REGION Network 5: Special Function Buttons Operator Control Allowed
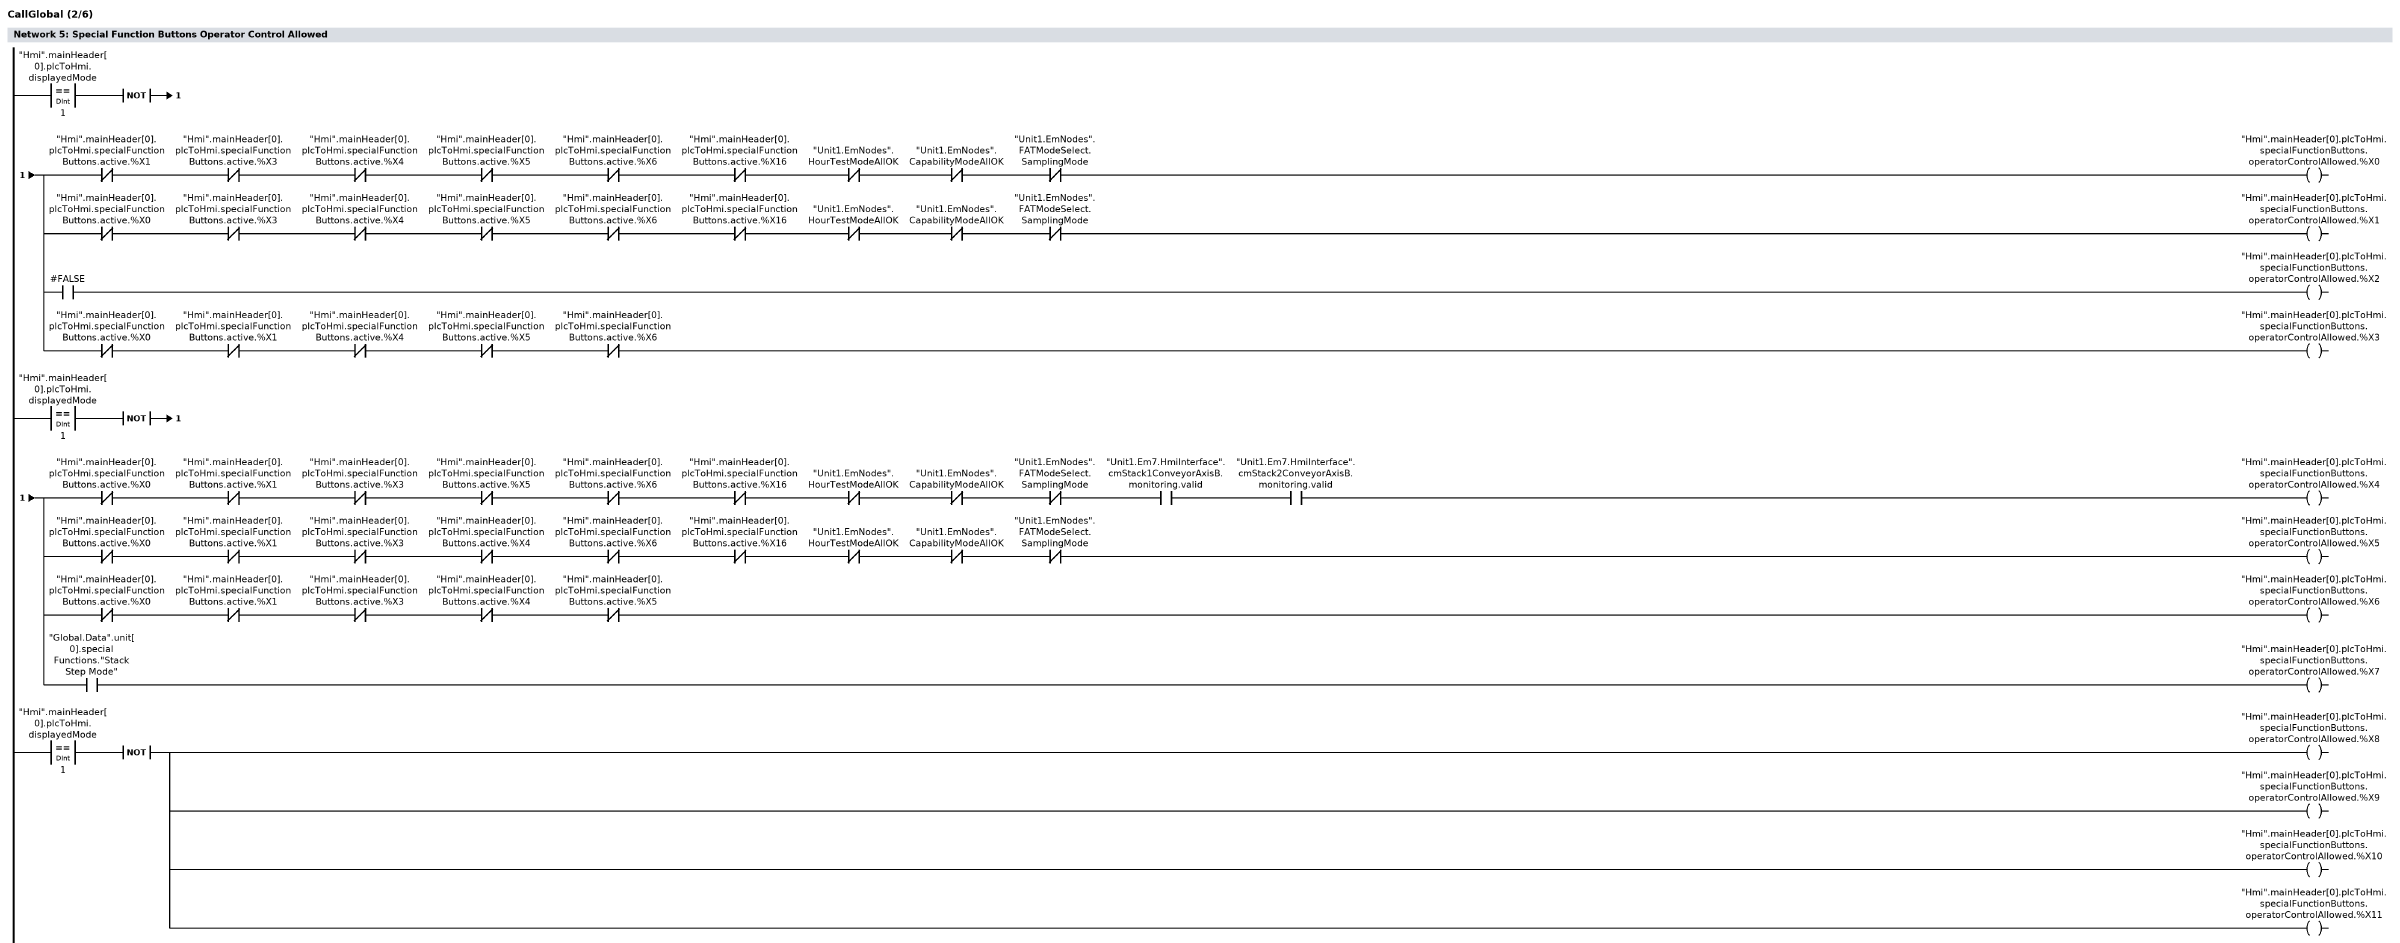
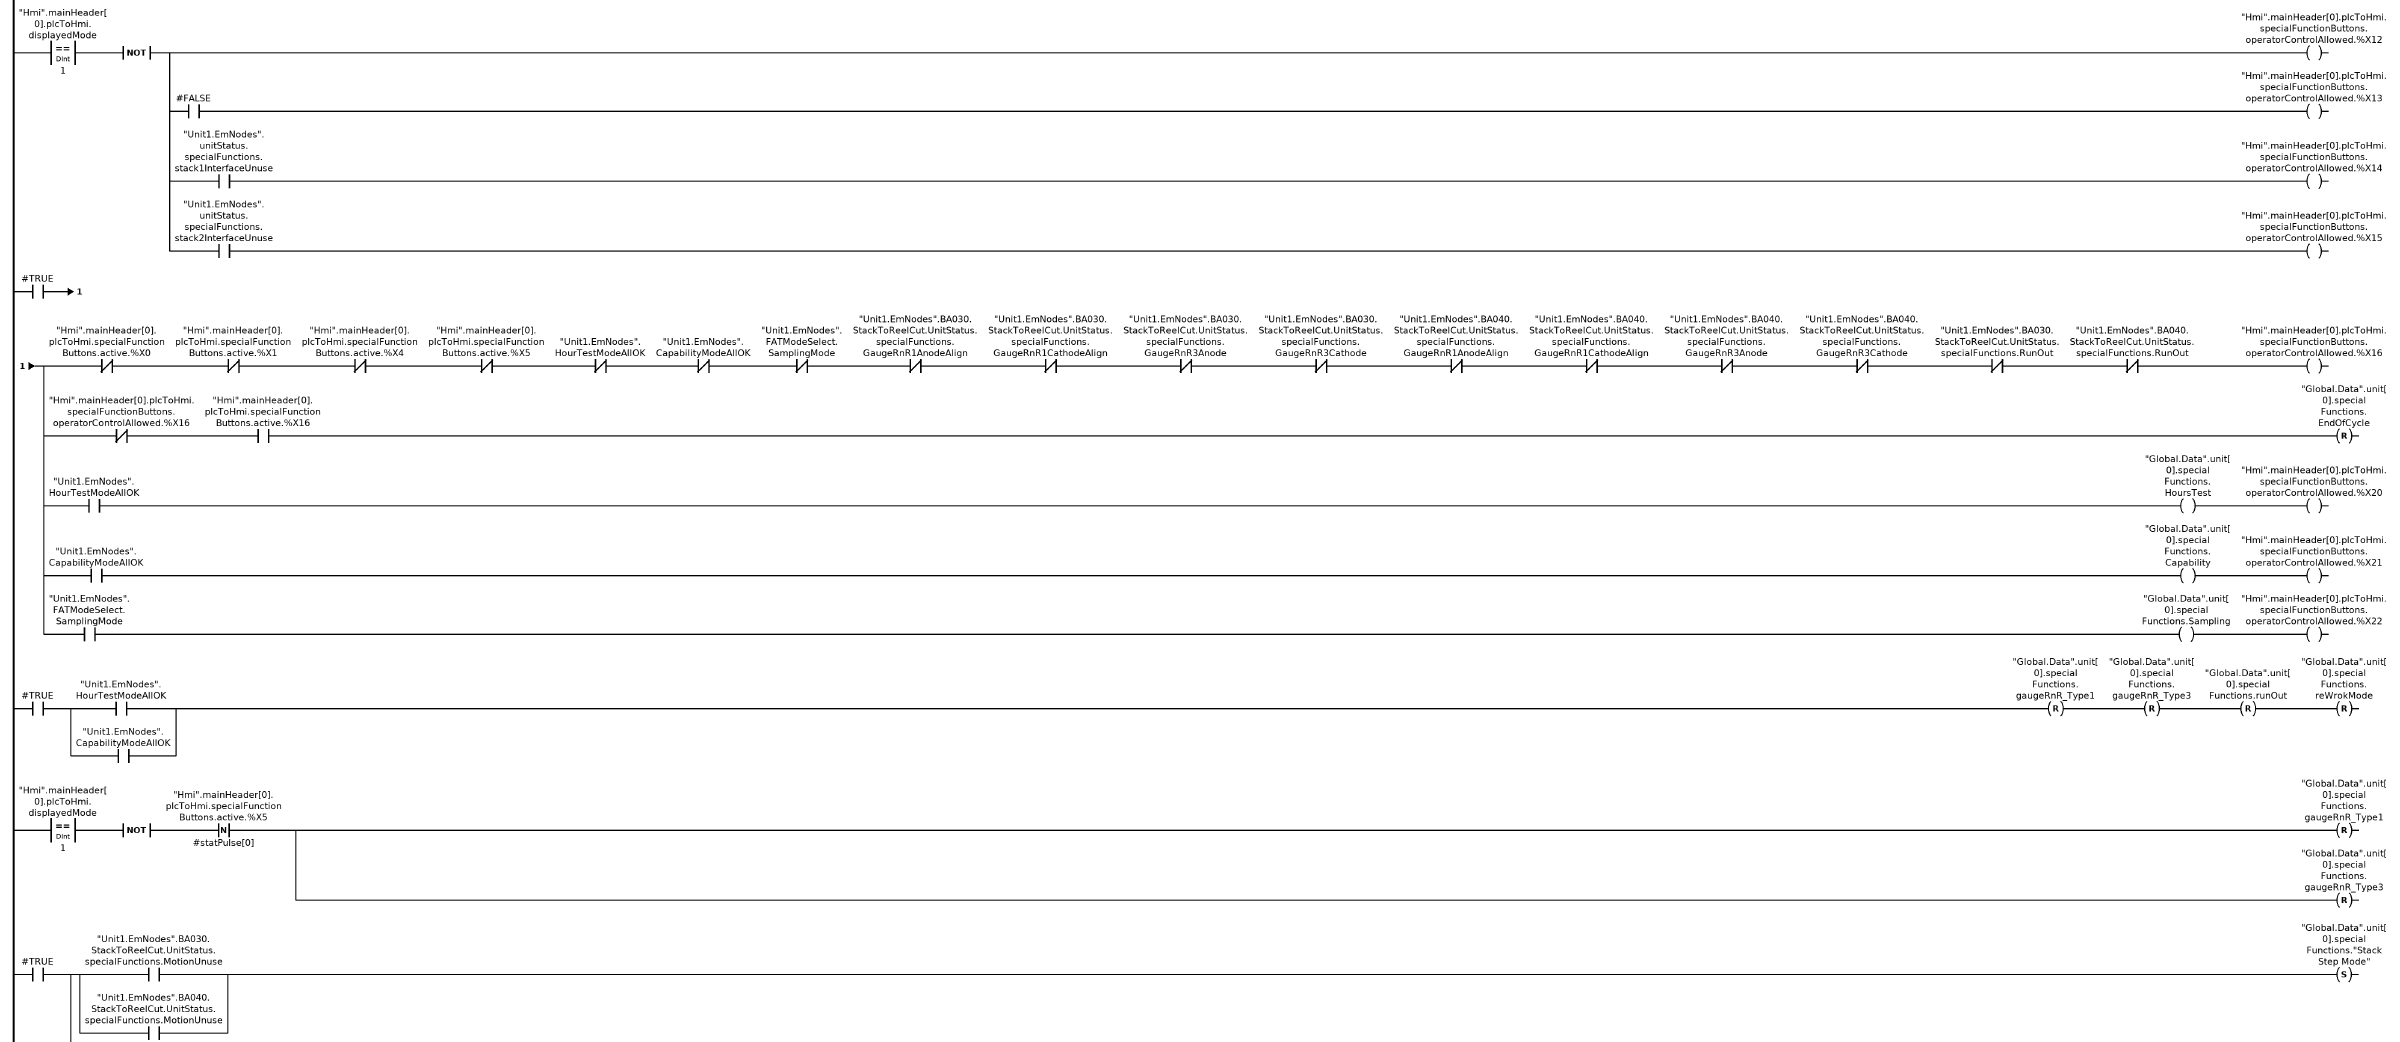
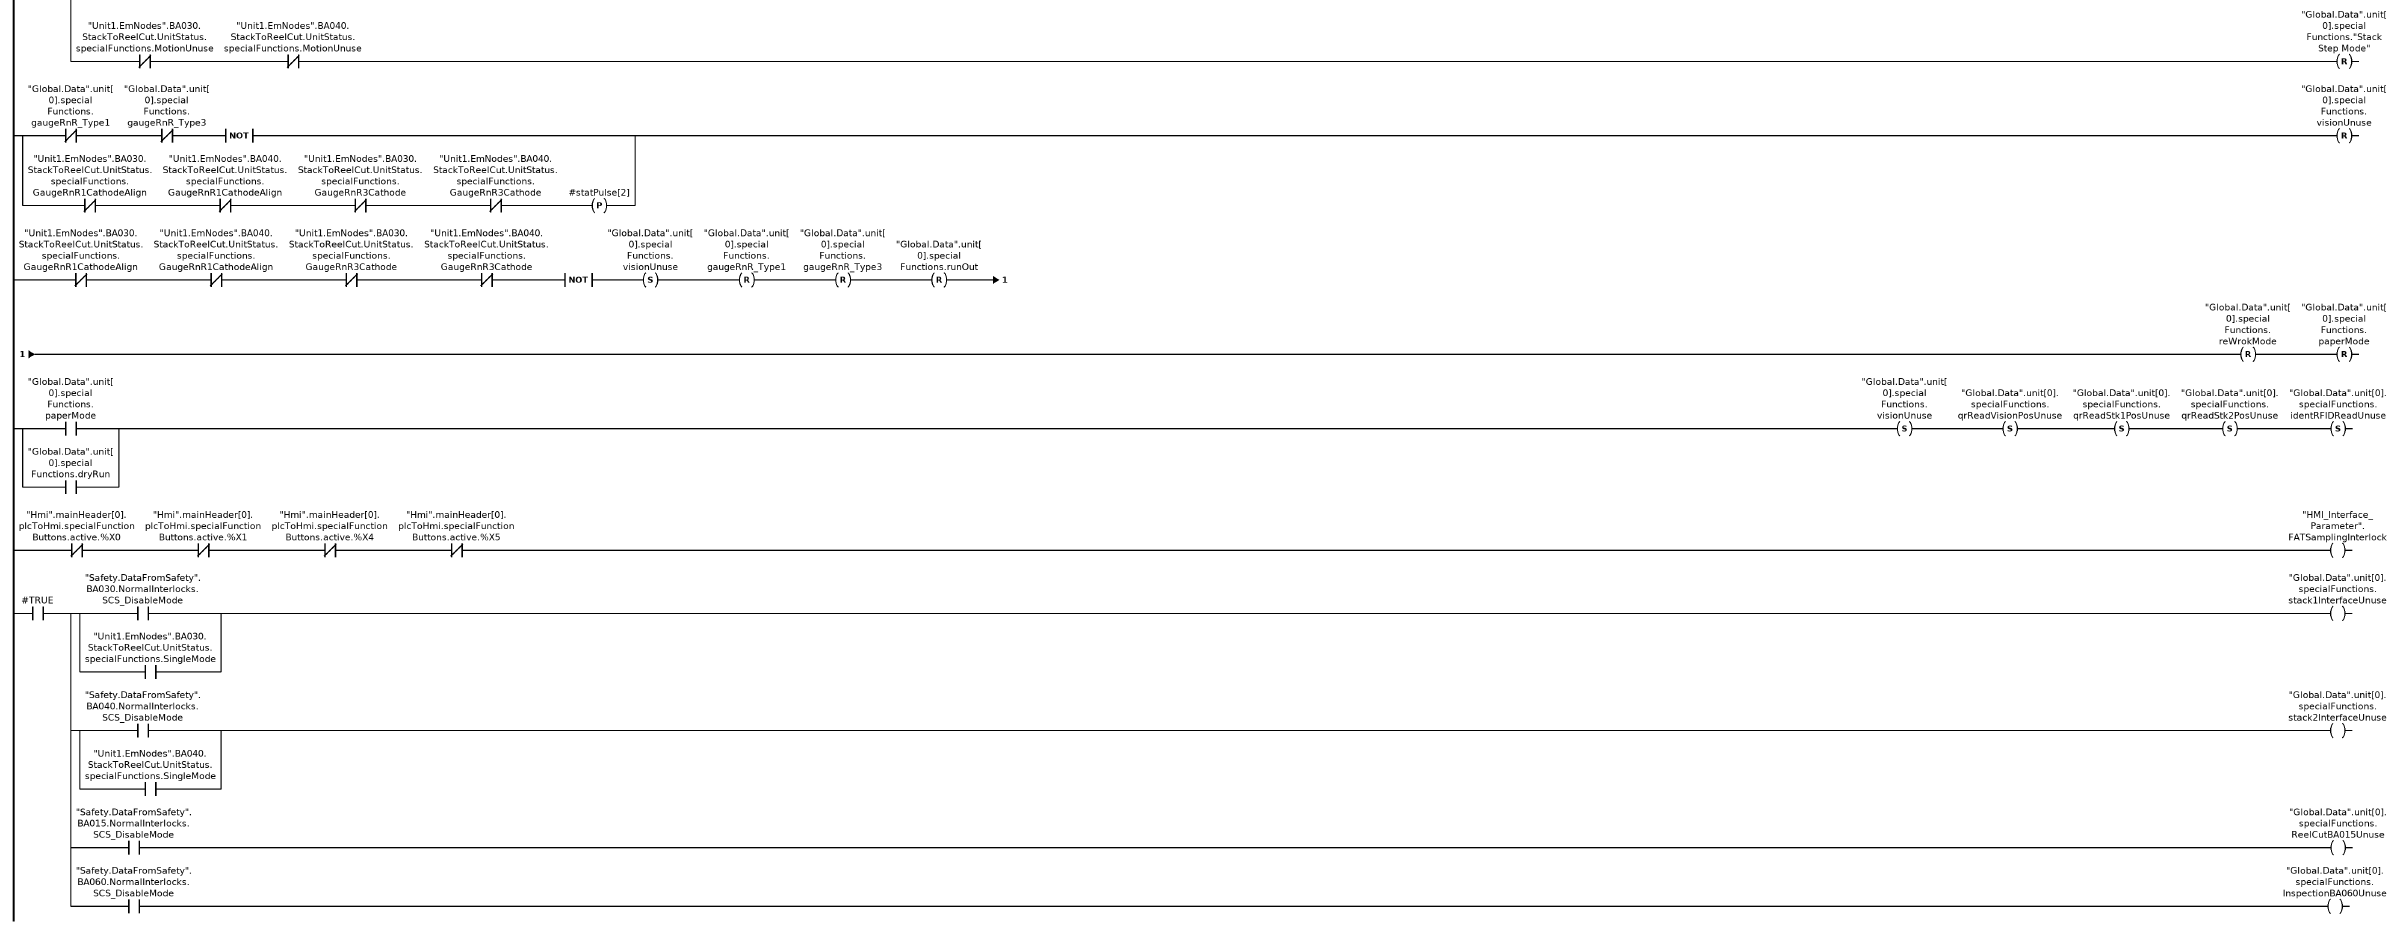
   RUNG wire#powerrail
      { S7_Templates := "SrcType := DInt" } EQ_Contact(in1 := "Hmi".mainHeader[0].plcToHmi.displayedMode, in2 := 1)
      Not()
      wire#w1
      I_Contact( "Hmi".mainHeader[0].plcToHmi.specialFunctionButtons.active.%X1 )
      I_Contact( "Hmi".mainHeader[0].plcToHmi.specialFunctionButtons.active.%X3 )
      I_Contact( "Hmi".mainHeader[0].plcToHmi.specialFunctionButtons.active.%X4 )
      I_Contact( "Hmi".mainHeader[0].plcToHmi.specialFunctionButtons.active.%X5 )
      I_Contact( "Hmi".mainHeader[0].plcToHmi.specialFunctionButtons.active.%X6 )
      I_Contact( "Hmi".mainHeader[0].plcToHmi.specialFunctionButtons.active.%X16 )
      I_Contact( "Unit1.EmNodes".HourTestModeAllOK )
      I_Contact( "Unit1.EmNodes".CapabilityModeAllOK )
      I_Contact( "Unit1.EmNodes".FATModeSelect.SamplingMode )
      Coil( "Hmi".mainHeader[0].plcToHmi.specialFunctionButtons.operatorControlAllowed.%X0 )
   END_RUNG
   RUNG wire#w1
      I_Contact( "Hmi".mainHeader[0].plcToHmi.specialFunctionButtons.active.%X0 )
      I_Contact( "Hmi".mainHeader[0].plcToHmi.specialFunctionButtons.active.%X3 )
      I_Contact( "Hmi".mainHeader[0].plcToHmi.specialFunctionButtons.active.%X4 )
      I_Contact( "Hmi".mainHeader[0].plcToHmi.specialFunctionButtons.active.%X5 )
      I_Contact( "Hmi".mainHeader[0].plcToHmi.specialFunctionButtons.active.%X6 )
      I_Contact( "Hmi".mainHeader[0].plcToHmi.specialFunctionButtons.active.%X16 )
      I_Contact( "Unit1.EmNodes".HourTestModeAllOK )
      I_Contact( "Unit1.EmNodes".CapabilityModeAllOK )
      I_Contact( "Unit1.EmNodes".FATModeSelect.SamplingMode )
      Coil( "Hmi".mainHeader[0].plcToHmi.specialFunctionButtons.operatorControlAllowed.%X1 )
   END_RUNG
   RUNG wire#w1
      Contact( #FALSE )
      Coil( "Hmi".mainHeader[0].plcToHmi.specialFunctionButtons.operatorControlAllowed.%X2 )
   END_RUNG
   RUNG wire#w1
      I_Contact( "Hmi".mainHeader[0].plcToHmi.specialFunctionButtons.active.%X0 )
      I_Contact( "Hmi".mainHeader[0].plcToHmi.specialFunctionButtons.active.%X1 )
      I_Contact( "Hmi".mainHeader[0].plcToHmi.specialFunctionButtons.active.%X4 )
      I_Contact( "Hmi".mainHeader[0].plcToHmi.specialFunctionButtons.active.%X5 )
      I_Contact( "Hmi".mainHeader[0].plcToHmi.specialFunctionButtons.active.%X6 )
      Coil( "Hmi".mainHeader[0].plcToHmi.specialFunctionButtons.operatorControlAllowed.%X3 )
   END_RUNG
   RUNG wire#powerrail
      { S7_Templates := "SrcType := DInt" } EQ_Contact(in1 := "Hmi".mainHeader[0].plcToHmi.displayedMode, in2 := 1)
      Not()
      wire#w2
      I_Contact( "Hmi".mainHeader[0].plcToHmi.specialFunctionButtons.active.%X0 )
      I_Contact( "Hmi".mainHeader[0].plcToHmi.specialFunctionButtons.active.%X1 )
      I_Contact( "Hmi".mainHeader[0].plcToHmi.specialFunctionButtons.active.%X3 )
      I_Contact( "Hmi".mainHeader[0].plcToHmi.specialFunctionButtons.active.%X5 )
      I_Contact( "Hmi".mainHeader[0].plcToHmi.specialFunctionButtons.active.%X6 )
      I_Contact( "Hmi".mainHeader[0].plcToHmi.specialFunctionButtons.active.%X16 )
      I_Contact( "Unit1.EmNodes".HourTestModeAllOK )
      I_Contact( "Unit1.EmNodes".CapabilityModeAllOK )
      I_Contact( "Unit1.EmNodes".FATModeSelect.SamplingMode )
      Contact( "Unit1.Em7.HmiInterface".cmStack1ConveyorAxisB.monitoring.valid )
      Contact( "Unit1.Em7.HmiInterface".cmStack2ConveyorAxisB.monitoring.valid )
      Coil( "Hmi".mainHeader[0].plcToHmi.specialFunctionButtons.operatorControlAllowed.%X4 )
   END_RUNG
   RUNG wire#w2
      I_Contact( "Hmi".mainHeader[0].plcToHmi.specialFunctionButtons.active.%X0 )
      I_Contact( "Hmi".mainHeader[0].plcToHmi.specialFunctionButtons.active.%X1 )
      I_Contact( "Hmi".mainHeader[0].plcToHmi.specialFunctionButtons.active.%X3 )
      I_Contact( "Hmi".mainHeader[0].plcToHmi.specialFunctionButtons.active.%X4 )
      I_Contact( "Hmi".mainHeader[0].plcToHmi.specialFunctionButtons.active.%X6 )
      I_Contact( "Hmi".mainHeader[0].plcToHmi.specialFunctionButtons.active.%X16 )
      I_Contact( "Unit1.EmNodes".HourTestModeAllOK )
      I_Contact( "Unit1.EmNodes".CapabilityModeAllOK )
      I_Contact( "Unit1.EmNodes".FATModeSelect.SamplingMode )
      Coil( "Hmi".mainHeader[0].plcToHmi.specialFunctionButtons.operatorControlAllowed.%X5 )
   END_RUNG
   RUNG wire#w2
      I_Contact( "Hmi".mainHeader[0].plcToHmi.specialFunctionButtons.active.%X0 )
      I_Contact( "Hmi".mainHeader[0].plcToHmi.specialFunctionButtons.active.%X1 )
      I_Contact( "Hmi".mainHeader[0].plcToHmi.specialFunctionButtons.active.%X3 )
      I_Contact( "Hmi".mainHeader[0].plcToHmi.specialFunctionButtons.active.%X4 )
      I_Contact( "Hmi".mainHeader[0].plcToHmi.specialFunctionButtons.active.%X5 )
      Coil( "Hmi".mainHeader[0].plcToHmi.specialFunctionButtons.operatorControlAllowed.%X6 )
   END_RUNG
   RUNG wire#w2
      Contact( "Global.Data".unit[0].specialFunctions."Stack Step Mode" )
      Coil( "Hmi".mainHeader[0].plcToHmi.specialFunctionButtons.operatorControlAllowed.%X7 )
   END_RUNG
   RUNG wire#powerrail
      { S7_Templates := "SrcType := DInt" } EQ_Contact(in1 := "Hmi".mainHeader[0].plcToHmi.displayedMode, in2 := 1)
      Not()
      wire#w3
      Coil( "Hmi".mainHeader[0].plcToHmi.specialFunctionButtons.operatorControlAllowed.%X8 )
   END_RUNG
   RUNG wire#w3
      Coil( "Hmi".mainHeader[0].plcToHmi.specialFunctionButtons.operatorControlAllowed.%X9 )
   END_RUNG
   RUNG wire#w3
      Coil( "Hmi".mainHeader[0].plcToHmi.specialFunctionButtons.operatorControlAllowed.%X10 )
   END_RUNG
   RUNG wire#w3
      Coil( "Hmi".mainHeader[0].plcToHmi.specialFunctionButtons.operatorControlAllowed.%X11 )
   END_RUNG
   RUNG wire#powerrail
      { S7_Templates := "SrcType := DInt" } EQ_Contact(in1 := "Hmi".mainHeader[0].plcToHmi.displayedMode, in2 := 1)
      Not()
      wire#w4
      Coil( "Hmi".mainHeader[0].plcToHmi.specialFunctionButtons.operatorControlAllowed.%X12 )
   END_RUNG
   RUNG wire#w4
      Contact( #FALSE )
      Coil( "Hmi".mainHeader[0].plcToHmi.specialFunctionButtons.operatorControlAllowed.%X13 )
   END_RUNG
   RUNG wire#w4
      Contact( "Unit1.EmNodes".unitStatus.specialFunctions.stack1InterfaceUnuse )
      Coil( "Hmi".mainHeader[0].plcToHmi.specialFunctionButtons.operatorControlAllowed.%X14 )
   END_RUNG
   RUNG wire#w4
      Contact( "Unit1.EmNodes".unitStatus.specialFunctions.stack2InterfaceUnuse )
      Coil( "Hmi".mainHeader[0].plcToHmi.specialFunctionButtons.operatorControlAllowed.%X15 )
   END_RUNG
   RUNG wire#powerrail
      Contact( #TRUE )
      wire#w5
      I_Contact( "Hmi".mainHeader[0].plcToHmi.specialFunctionButtons.active.%X0 )
      I_Contact( "Hmi".mainHeader[0].plcToHmi.specialFunctionButtons.active.%X1 )
      I_Contact( "Hmi".mainHeader[0].plcToHmi.specialFunctionButtons.active.%X4 )
      I_Contact( "Hmi".mainHeader[0].plcToHmi.specialFunctionButtons.active.%X5 )
      I_Contact( "Unit1.EmNodes".HourTestModeAllOK )
      I_Contact( "Unit1.EmNodes".CapabilityModeAllOK )
      I_Contact( "Unit1.EmNodes".FATModeSelect.SamplingMode )
      I_Contact( "Unit1.EmNodes".BA030.StackToReelCut.UnitStatus.specialFunctions.GaugeRnR1AnodeAlign )
      I_Contact( "Unit1.EmNodes".BA030.StackToReelCut.UnitStatus.specialFunctions.GaugeRnR1CathodeAlign )
      I_Contact( "Unit1.EmNodes".BA030.StackToReelCut.UnitStatus.specialFunctions.GaugeRnR3Anode )
      I_Contact( "Unit1.EmNodes".BA030.StackToReelCut.UnitStatus.specialFunctions.GaugeRnR3Cathode )
      I_Contact( "Unit1.EmNodes".BA040.StackToReelCut.UnitStatus.specialFunctions.GaugeRnR1AnodeAlign )
      I_Contact( "Unit1.EmNodes".BA040.StackToReelCut.UnitStatus.specialFunctions.GaugeRnR1CathodeAlign )
      I_Contact( "Unit1.EmNodes".BA040.StackToReelCut.UnitStatus.specialFunctions.GaugeRnR3Anode )
      I_Contact( "Unit1.EmNodes".BA040.StackToReelCut.UnitStatus.specialFunctions.GaugeRnR3Cathode )
      I_Contact( "Unit1.EmNodes".BA030.StackToReelCut.UnitStatus.specialFunctions.RunOut )
      I_Contact( "Unit1.EmNodes".BA040.StackToReelCut.UnitStatus.specialFunctions.RunOut )
      Coil( "Hmi".mainHeader[0].plcToHmi.specialFunctionButtons.operatorControlAllowed.%X16 )
   END_RUNG
   RUNG wire#w5
      I_Contact( "Hmi".mainHeader[0].plcToHmi.specialFunctionButtons.operatorControlAllowed.%X16 )
      Contact( "Hmi".mainHeader[0].plcToHmi.specialFunctionButtons.active.%X16 )
      R_Coil( "Global.Data".unit[0].specialFunctions.EndOfCycle )
   END_RUNG
   RUNG wire#w5
      Contact( "Unit1.EmNodes".HourTestModeAllOK )
      Coil( "Global.Data".unit[0].specialFunctions.HoursTest )
      Coil( "Hmi".mainHeader[0].plcToHmi.specialFunctionButtons.operatorControlAllowed.%X20 )
   END_RUNG
   RUNG wire#w5
      Contact( "Unit1.EmNodes".CapabilityModeAllOK )
      Coil( "Global.Data".unit[0].specialFunctions.Capability )
      Coil( "Hmi".mainHeader[0].plcToHmi.specialFunctionButtons.operatorControlAllowed.%X21 )
   END_RUNG
   RUNG wire#w5
      Contact( "Unit1.EmNodes".FATModeSelect.SamplingMode )
      Coil( "Global.Data".unit[0].specialFunctions.Sampling )
      Coil( "Hmi".mainHeader[0].plcToHmi.specialFunctionButtons.operatorControlAllowed.%X22 )
   END_RUNG
   RUNG wire#powerrail
      Contact( #TRUE )
      wire#w6
      Contact( "Unit1.EmNodes".HourTestModeAllOK )
      wire#w7
      R_Coil( "Global.Data".unit[0].specialFunctions.gaugeRnR_Type1 )
      R_Coil( "Global.Data".unit[0].specialFunctions.gaugeRnR_Type3 )
      R_Coil( "Global.Data".unit[0].specialFunctions.runOut )
      R_Coil( "Global.Data".unit[0].specialFunctions.reWrokMode )
   END_RUNG
   RUNG wire#w6
      Contact( "Unit1.EmNodes".CapabilityModeAllOK )
   END_RUNG wire#w7
   RUNG wire#powerrail
      { S7_Templates := "SrcType := DInt" } EQ_Contact(in1 := "Hmi".mainHeader[0].plcToHmi.displayedMode, in2 := 1)
      Not()
      N_Contact(operand := "Hmi".mainHeader[0].plcToHmi.specialFunctionButtons.active.%X5, bit := #statPulse[0])
      wire#w8
      R_Coil( "Global.Data".unit[0].specialFunctions.gaugeRnR_Type1 )
   END_RUNG
   RUNG wire#w8
      R_Coil( "Global.Data".unit[0].specialFunctions.gaugeRnR_Type3 )
   END_RUNG
   RUNG wire#powerrail
      Contact( #TRUE )
      wire#w9
      Contact( "Unit1.EmNodes".BA030.StackToReelCut.UnitStatus.specialFunctions.MotionUnuse )
      wire#w10
      S_Coil( "Global.Data".unit[0].specialFunctions."Stack Step Mode" )
   END_RUNG
   RUNG wire#w9
      Contact( "Unit1.EmNodes".BA040.StackToReelCut.UnitStatus.specialFunctions.MotionUnuse )
   END_RUNG wire#w10
   RUNG wire#w9
      I_Contact( "Unit1.EmNodes".BA030.StackToReelCut.UnitStatus.specialFunctions.MotionUnuse )
      I_Contact( "Unit1.EmNodes".BA040.StackToReelCut.UnitStatus.specialFunctions.MotionUnuse )
      R_Coil( "Global.Data".unit[0].specialFunctions."Stack Step Mode" )
   END_RUNG
   RUNG wire#powerrail
      I_Contact( "Global.Data".unit[0].specialFunctions.gaugeRnR_Type1 )
      I_Contact( "Global.Data".unit[0].specialFunctions.gaugeRnR_Type3 )
      Not()
      wire#w11
      R_Coil( "Global.Data".unit[0].specialFunctions.visionUnuse )
   END_RUNG
   RUNG wire#powerrail
      I_Contact( "Unit1.EmNodes".BA030.StackToReelCut.UnitStatus.specialFunctions.GaugeRnR1CathodeAlign )
      I_Contact( "Unit1.EmNodes".BA040.StackToReelCut.UnitStatus.specialFunctions.GaugeRnR1CathodeAlign )
      I_Contact( "Unit1.EmNodes".BA030.StackToReelCut.UnitStatus.specialFunctions.GaugeRnR3Cathode )
      I_Contact( "Unit1.EmNodes".BA040.StackToReelCut.UnitStatus.specialFunctions.GaugeRnR3Cathode )
      P_Trig( #statPulse[2] )
   END_RUNG wire#w11
   RUNG wire#powerrail
      I_Contact( "Unit1.EmNodes".BA030.StackToReelCut.UnitStatus.specialFunctions.GaugeRnR1CathodeAlign )
      I_Contact( "Unit1.EmNodes".BA040.StackToReelCut.UnitStatus.specialFunctions.GaugeRnR1CathodeAlign )
      I_Contact( "Unit1.EmNodes".BA030.StackToReelCut.UnitStatus.specialFunctions.GaugeRnR3Cathode )
      I_Contact( "Unit1.EmNodes".BA040.StackToReelCut.UnitStatus.specialFunctions.GaugeRnR3Cathode )
      Not()
      S_Coil( "Global.Data".unit[0].specialFunctions.visionUnuse )
      R_Coil( "Global.Data".unit[0].specialFunctions.gaugeRnR_Type1 )
      R_Coil( "Global.Data".unit[0].specialFunctions.gaugeRnR_Type3 )
      R_Coil( "Global.Data".unit[0].specialFunctions.runOut )
      R_Coil( "Global.Data".unit[0].specialFunctions.reWrokMode )
      R_Coil( "Global.Data".unit[0].specialFunctions.paperMode )
   END_RUNG
   RUNG wire#powerrail
      Contact( "Global.Data".unit[0].specialFunctions.paperMode )
      wire#w12
      S_Coil( "Global.Data".unit[0].specialFunctions.visionUnuse )
      S_Coil( "Global.Data".unit[0].specialFunctions.qrReadVisionPosUnuse )
      S_Coil( "Global.Data".unit[0].specialFunctions.qrReadStk1PosUnuse )
      S_Coil( "Global.Data".unit[0].specialFunctions.qrReadStk2PosUnuse )
      S_Coil( "Global.Data".unit[0].specialFunctions.identRFIDReadUnuse )
   END_RUNG
   RUNG wire#powerrail
      Contact( "Global.Data".unit[0].specialFunctions.dryRun )
   END_RUNG wire#w12
   RUNG wire#powerrail
      I_Contact( "Hmi".mainHeader[0].plcToHmi.specialFunctionButtons.active.%X0 )
      I_Contact( "Hmi".mainHeader[0].plcToHmi.specialFunctionButtons.active.%X1 )
      I_Contact( "Hmi".mainHeader[0].plcToHmi.specialFunctionButtons.active.%X4 )
      I_Contact( "Hmi".mainHeader[0].plcToHmi.specialFunctionButtons.active.%X5 )
      Coil( "HMI_Interface_Parameter".FATSamplingInterlock )
   END_RUNG
   RUNG wire#powerrail
      Contact( #TRUE )
      wire#w13
      Contact( "Safety.DataFromSafety".BA030.NormalInterlocks.SCS_DisableMode )
      wire#w14
      Coil( "Global.Data".unit[0].specialFunctions.stack1InterfaceUnuse )
   END_RUNG
   RUNG wire#w13
      Contact( "Unit1.EmNodes".BA030.StackToReelCut.UnitStatus.specialFunctions.SingleMode )
   END_RUNG wire#w14
   RUNG wire#w13
      Contact( "Safety.DataFromSafety".BA040.NormalInterlocks.SCS_DisableMode )
      wire#w15
      Coil( "Global.Data".unit[0].specialFunctions.stack2InterfaceUnuse )
   END_RUNG
   RUNG wire#w13
      Contact( "Unit1.EmNodes".BA040.StackToReelCut.UnitStatus.specialFunctions.SingleMode )
   END_RUNG wire#w15
   RUNG wire#w13
      Contact( "Safety.DataFromSafety".BA015.NormalInterlocks.SCS_DisableMode )
      Coil( "Global.Data".unit[0].specialFunctions.ReelCutBA015Unuse )
   END_RUNG
   RUNG wire#w13
      Contact( "Safety.DataFromSafety".BA060.NormalInterlocks.SCS_DisableMode )
      Coil( "Global.Data".unit[0].specialFunctions.InspectionBA060Unuse )
   END_RUNG
   // the same network as SCL:
   #_w1 := NOT ("Hmi".mainHeader[0].plcToHmi.displayedMode = 1);
   "Hmi".mainHeader[0].plcToHmi.specialFunctionButtons.operatorControlAllowed.%X0 := #_w1 AND NOT "Hmi".mainHeader[0].plcToHmi.specialFunctionButtons.active.%X1 AND NOT "Hmi".mainHeader[0].plcToHmi.specialFunctionButtons.active.%X3 AND NOT "Hmi".mainHeader[0].plcToHmi.specialFunctionButtons.active.%X4 AND NOT "Hmi".mainHeader[0].plcToHmi.specialFunctionButtons.active.%X5 AND NOT "Hmi".mainHeader[0].plcToHmi.specialFunctionButtons.active.%X6 AND NOT "Hmi".mainHeader[0].plcToHmi.specialFunctionButtons.active.%X16 AND NOT "Unit1.EmNodes".HourTestModeAllOK AND NOT "Unit1.EmNodes".CapabilityModeAllOK AND NOT "Unit1.EmNodes".FATModeSelect.SamplingMode;
   "Hmi".mainHeader[0].plcToHmi.specialFunctionButtons.operatorControlAllowed.%X1 := #_w1 AND NOT "Hmi".mainHeader[0].plcToHmi.specialFunctionButtons.active.%X0 AND NOT "Hmi".mainHeader[0].plcToHmi.specialFunctionButtons.active.%X3 AND NOT "Hmi".mainHeader[0].plcToHmi.specialFunctionButtons.active.%X4 AND NOT "Hmi".mainHeader[0].plcToHmi.specialFunctionButtons.active.%X5 AND NOT "Hmi".mainHeader[0].plcToHmi.specialFunctionButtons.active.%X6 AND NOT "Hmi".mainHeader[0].plcToHmi.specialFunctionButtons.active.%X16 AND NOT "Unit1.EmNodes".HourTestModeAllOK AND NOT "Unit1.EmNodes".CapabilityModeAllOK AND NOT "Unit1.EmNodes".FATModeSelect.SamplingMode;
   "Hmi".mainHeader[0].plcToHmi.specialFunctionButtons.operatorControlAllowed.%X2 := #_w1 AND #FALSE;
   "Hmi".mainHeader[0].plcToHmi.specialFunctionButtons.operatorControlAllowed.%X3 := #_w1 AND NOT "Hmi".mainHeader[0].plcToHmi.specialFunctionButtons.active.%X0 AND NOT "Hmi".mainHeader[0].plcToHmi.specialFunctionButtons.active.%X1 AND NOT "Hmi".mainHeader[0].plcToHmi.specialFunctionButtons.active.%X4 AND NOT "Hmi".mainHeader[0].plcToHmi.specialFunctionButtons.active.%X5 AND NOT "Hmi".mainHeader[0].plcToHmi.specialFunctionButtons.active.%X6;
   #_w2 := NOT ("Hmi".mainHeader[0].plcToHmi.displayedMode = 1);
   "Hmi".mainHeader[0].plcToHmi.specialFunctionButtons.operatorControlAllowed.%X4 := #_w2 AND NOT "Hmi".mainHeader[0].plcToHmi.specialFunctionButtons.active.%X0 AND NOT "Hmi".mainHeader[0].plcToHmi.specialFunctionButtons.active.%X1 AND NOT "Hmi".mainHeader[0].plcToHmi.specialFunctionButtons.active.%X3 AND NOT "Hmi".mainHeader[0].plcToHmi.specialFunctionButtons.active.%X5 AND NOT "Hmi".mainHeader[0].plcToHmi.specialFunctionButtons.active.%X6 AND NOT "Hmi".mainHeader[0].plcToHmi.specialFunctionButtons.active.%X16 AND NOT "Unit1.EmNodes".HourTestModeAllOK AND NOT "Unit1.EmNodes".CapabilityModeAllOK AND NOT "Unit1.EmNodes".FATModeSelect.SamplingMode AND "Unit1.Em7.HmiInterface".cmStack1ConveyorAxisB.monitoring.valid AND "Unit1.Em7.HmiInterface".cmStack2ConveyorAxisB.monitoring.valid;
   "Hmi".mainHeader[0].plcToHmi.specialFunctionButtons.operatorControlAllowed.%X5 := #_w2 AND NOT "Hmi".mainHeader[0].plcToHmi.specialFunctionButtons.active.%X0 AND NOT "Hmi".mainHeader[0].plcToHmi.specialFunctionButtons.active.%X1 AND NOT "Hmi".mainHeader[0].plcToHmi.specialFunctionButtons.active.%X3 AND NOT "Hmi".mainHeader[0].plcToHmi.specialFunctionButtons.active.%X4 AND NOT "Hmi".mainHeader[0].plcToHmi.specialFunctionButtons.active.%X6 AND NOT "Hmi".mainHeader[0].plcToHmi.specialFunctionButtons.active.%X16 AND NOT "Unit1.EmNodes".HourTestModeAllOK AND NOT "Unit1.EmNodes".CapabilityModeAllOK AND NOT "Unit1.EmNodes".FATModeSelect.SamplingMode;
   "Hmi".mainHeader[0].plcToHmi.specialFunctionButtons.operatorControlAllowed.%X6 := #_w2 AND NOT "Hmi".mainHeader[0].plcToHmi.specialFunctionButtons.active.%X0 AND NOT "Hmi".mainHeader[0].plcToHmi.specialFunctionButtons.active.%X1 AND NOT "Hmi".mainHeader[0].plcToHmi.specialFunctionButtons.active.%X3 AND NOT "Hmi".mainHeader[0].plcToHmi.specialFunctionButtons.active.%X4 AND NOT "Hmi".mainHeader[0].plcToHmi.specialFunctionButtons.active.%X5;
   "Hmi".mainHeader[0].plcToHmi.specialFunctionButtons.operatorControlAllowed.%X7 := #_w2 AND "Global.Data".unit[0].specialFunctions."Stack Step Mode";
   #_w3 := NOT ("Hmi".mainHeader[0].plcToHmi.displayedMode = 1);
   "Hmi".mainHeader[0].plcToHmi.specialFunctionButtons.operatorControlAllowed.%X8 := NOT ("Hmi".mainHeader[0].plcToHmi.displayedMode = 1);
   "Hmi".mainHeader[0].plcToHmi.specialFunctionButtons.operatorControlAllowed.%X9 := #_w3;
   "Hmi".mainHeader[0].plcToHmi.specialFunctionButtons.operatorControlAllowed.%X10 := #_w3;
   "Hmi".mainHeader[0].plcToHmi.specialFunctionButtons.operatorControlAllowed.%X11 := #_w3;
   #_w4 := NOT ("Hmi".mainHeader[0].plcToHmi.displayedMode = 1);
   "Hmi".mainHeader[0].plcToHmi.specialFunctionButtons.operatorControlAllowed.%X12 := NOT ("Hmi".mainHeader[0].plcToHmi.displayedMode = 1);
   "Hmi".mainHeader[0].plcToHmi.specialFunctionButtons.operatorControlAllowed.%X13 := #_w4 AND #FALSE;
   "Hmi".mainHeader[0].plcToHmi.specialFunctionButtons.operatorControlAllowed.%X14 := #_w4 AND "Unit1.EmNodes".unitStatus.specialFunctions.stack1InterfaceUnuse;
   "Hmi".mainHeader[0].plcToHmi.specialFunctionButtons.operatorControlAllowed.%X15 := #_w4 AND "Unit1.EmNodes".unitStatus.specialFunctions.stack2InterfaceUnuse;
   "Hmi".mainHeader[0].plcToHmi.specialFunctionButtons.operatorControlAllowed.%X16 := #TRUE AND NOT "Hmi".mainHeader[0].plcToHmi.specialFunctionButtons.active.%X0 AND NOT "Hmi".mainHeader[0].plcToHmi.specialFunctionButtons.active.%X1 AND NOT "Hmi".mainHeader[0].plcToHmi.specialFunctionButtons.active.%X4 AND NOT "Hmi".mainHeader[0].plcToHmi.specialFunctionButtons.active.%X5 AND NOT "Unit1.EmNodes".HourTestModeAllOK AND NOT "Unit1.EmNodes".CapabilityModeAllOK AND NOT "Unit1.EmNodes".FATModeSelect.SamplingMode AND NOT "Unit1.EmNodes".BA030.StackToReelCut.UnitStatus.specialFunctions.GaugeRnR1AnodeAlign AND NOT "Unit1.EmNodes".BA030.StackToReelCut.UnitStatus.specialFunctions.GaugeRnR1CathodeAlign AND NOT "Unit1.EmNodes".BA030.StackToReelCut.UnitStatus.specialFunctions.GaugeRnR3Anode AND NOT "Unit1.EmNodes".BA030.StackToReelCut.UnitStatus.specialFunctions.GaugeRnR3Cathode AND NOT "Unit1.EmNodes".BA040.StackToReelCut.UnitStatus.specialFunctions.GaugeRnR1AnodeAlign AND NOT "Unit1.EmNodes".BA040.StackToReelCut.UnitStatus.specialFunctions.GaugeRnR1CathodeAlign AND NOT "Unit1.EmNodes".BA040.StackToReelCut.UnitStatus.specialFunctions.GaugeRnR3Anode AND NOT "Unit1.EmNodes".BA040.StackToReelCut.UnitStatus.specialFunctions.GaugeRnR3Cathode AND NOT "Unit1.EmNodes".BA030.StackToReelCut.UnitStatus.specialFunctions.RunOut AND NOT "Unit1.EmNodes".BA040.StackToReelCut.UnitStatus.specialFunctions.RunOut;
   IF #TRUE AND NOT "Hmi".mainHeader[0].plcToHmi.specialFunctionButtons.operatorControlAllowed.%X16 AND "Hmi".mainHeader[0].plcToHmi.specialFunctionButtons.active.%X16 THEN
       "Global.Data".unit[0].specialFunctions.EndOfCycle := FALSE;
   END_IF;
   "Global.Data".unit[0].specialFunctions.HoursTest := #TRUE AND "Unit1.EmNodes".HourTestModeAllOK;
   "Hmi".mainHeader[0].plcToHmi.specialFunctionButtons.operatorControlAllowed.%X20 := #TRUE AND "Unit1.EmNodes".HourTestModeAllOK;
   "Global.Data".unit[0].specialFunctions.Capability := #TRUE AND "Unit1.EmNodes".CapabilityModeAllOK;
   "Hmi".mainHeader[0].plcToHmi.specialFunctionButtons.operatorControlAllowed.%X21 := #TRUE AND "Unit1.EmNodes".CapabilityModeAllOK;
   "Global.Data".unit[0].specialFunctions.Sampling := #TRUE AND "Unit1.EmNodes".FATModeSelect.SamplingMode;
   "Hmi".mainHeader[0].plcToHmi.specialFunctionButtons.operatorControlAllowed.%X22 := #TRUE AND "Unit1.EmNodes".FATModeSelect.SamplingMode;
   IF #TRUE AND ("Unit1.EmNodes".HourTestModeAllOK OR "Unit1.EmNodes".CapabilityModeAllOK) THEN
       "Global.Data".unit[0].specialFunctions.gaugeRnR_Type1 := FALSE;
       "Global.Data".unit[0].specialFunctions.gaugeRnR_Type3 := FALSE;
       "Global.Data".unit[0].specialFunctions.runOut := FALSE;
       "Global.Data".unit[0].specialFunctions.reWrokMode := FALSE;
   END_IF;
   #_w5 := NOT ("Hmi".mainHeader[0].plcToHmi.displayedMode = 1) AND NOT "Hmi".mainHeader[0].plcToHmi.specialFunctionButtons.active.%X5 AND #statPulse[0];   // falling edge of "Hmi".mainHeader[0].plcToHmi.specialFunctionButtons.active.%X5
   #statPulse[0] := "Hmi".mainHeader[0].plcToHmi.specialFunctionButtons.active.%X5;
   IF #_w5 THEN
       "Global.Data".unit[0].specialFunctions.gaugeRnR_Type1 := FALSE;
       "Global.Data".unit[0].specialFunctions.gaugeRnR_Type3 := FALSE;
   END_IF;
   IF #TRUE AND ("Unit1.EmNodes".BA030.StackToReelCut.UnitStatus.specialFunctions.MotionUnuse OR "Unit1.EmNodes".BA040.StackToReelCut.UnitStatus.specialFunctions.MotionUnuse) THEN
       "Global.Data".unit[0].specialFunctions."Stack Step Mode" := TRUE;
   END_IF;
   IF #TRUE AND NOT "Unit1.EmNodes".BA030.StackToReelCut.UnitStatus.specialFunctions.MotionUnuse AND NOT "Unit1.EmNodes".BA040.StackToReelCut.UnitStatus.specialFunctions.MotionUnuse THEN
       "Global.Data".unit[0].specialFunctions."Stack Step Mode" := FALSE;
   END_IF;
   #_w6 := NOT "Unit1.EmNodes".BA030.StackToReelCut.UnitStatus.specialFunctions.GaugeRnR1CathodeAlign AND NOT "Unit1.EmNodes".BA040.StackToReelCut.UnitStatus.specialFunctions.GaugeRnR1CathodeAlign AND NOT "Unit1.EmNodes".BA030.StackToReelCut.UnitStatus.specialFunctions.GaugeRnR3Cathode AND NOT "Unit1.EmNodes".BA040.StackToReelCut.UnitStatus.specialFunctions.GaugeRnR3Cathode;
   #_w7 := #_w6 AND NOT #statPulse[2];   // rising edge
   #statPulse[2] := #_w6;
   IF NOT (NOT "Global.Data".unit[0].specialFunctions.gaugeRnR_Type1 AND NOT "Global.Data".unit[0].specialFunctions.gaugeRnR_Type3) OR #_w7 THEN
       "Global.Data".unit[0].specialFunctions.visionUnuse := FALSE;
   END_IF;
   IF NOT (NOT "Unit1.EmNodes".BA030.StackToReelCut.UnitStatus.specialFunctions.GaugeRnR1CathodeAlign AND NOT "Unit1.EmNodes".BA040.StackToReelCut.UnitStatus.specialFunctions.GaugeRnR1CathodeAlign AND NOT "Unit1.EmNodes".BA030.StackToReelCut.UnitStatus.specialFunctions.GaugeRnR3Cathode AND NOT "Unit1.EmNodes".BA040.StackToReelCut.UnitStatus.specialFunctions.GaugeRnR3Cathode) THEN
       "Global.Data".unit[0].specialFunctions.visionUnuse := TRUE;
       "Global.Data".unit[0].specialFunctions.gaugeRnR_Type1 := FALSE;
       "Global.Data".unit[0].specialFunctions.gaugeRnR_Type3 := FALSE;
       "Global.Data".unit[0].specialFunctions.runOut := FALSE;
       "Global.Data".unit[0].specialFunctions.reWrokMode := FALSE;
       "Global.Data".unit[0].specialFunctions.paperMode := FALSE;
   END_IF;
   #_w8 := "Global.Data".unit[0].specialFunctions.paperMode OR "Global.Data".unit[0].specialFunctions.dryRun;
   IF #_w8 THEN
       "Global.Data".unit[0].specialFunctions.visionUnuse := TRUE;
       "Global.Data".unit[0].specialFunctions.qrReadVisionPosUnuse := TRUE;
       "Global.Data".unit[0].specialFunctions.qrReadStk1PosUnuse := TRUE;
       "Global.Data".unit[0].specialFunctions.qrReadStk2PosUnuse := TRUE;
       "Global.Data".unit[0].specialFunctions.identRFIDReadUnuse := TRUE;
   END_IF;
   "HMI_Interface_Parameter".FATSamplingInterlock := NOT "Hmi".mainHeader[0].plcToHmi.specialFunctionButtons.active.%X0 AND NOT "Hmi".mainHeader[0].plcToHmi.specialFunctionButtons.active.%X1 AND NOT "Hmi".mainHeader[0].plcToHmi.specialFunctionButtons.active.%X4 AND NOT "Hmi".mainHeader[0].plcToHmi.specialFunctionButtons.active.%X5;
   "Global.Data".unit[0].specialFunctions.stack1InterfaceUnuse := #TRUE AND ("Safety.DataFromSafety".BA030.NormalInterlocks.SCS_DisableMode OR "Unit1.EmNodes".BA030.StackToReelCut.UnitStatus.specialFunctions.SingleMode);
   "Global.Data".unit[0].specialFunctions.stack2InterfaceUnuse := #TRUE AND ("Safety.DataFromSafety".BA040.NormalInterlocks.SCS_DisableMode OR "Unit1.EmNodes".BA040.StackToReelCut.UnitStatus.specialFunctions.SingleMode);
   "Global.Data".unit[0].specialFunctions.ReelCutBA015Unuse := #TRUE AND "Safety.DataFromSafety".BA015.NormalInterlocks.SCS_DisableMode;
   "Global.Data".unit[0].specialFunctions.InspectionBA060Unuse := #TRUE AND "Safety.DataFromSafety".BA060.NormalInterlocks.SCS_DisableMode;
END_REGION

REGION Network 6: HMI Control Header
   // Read the input from the control header in the HMI an distribute information to the according units. Vice versa, summarize the unit information and provide it to the control header to display e.g. the modes and states.
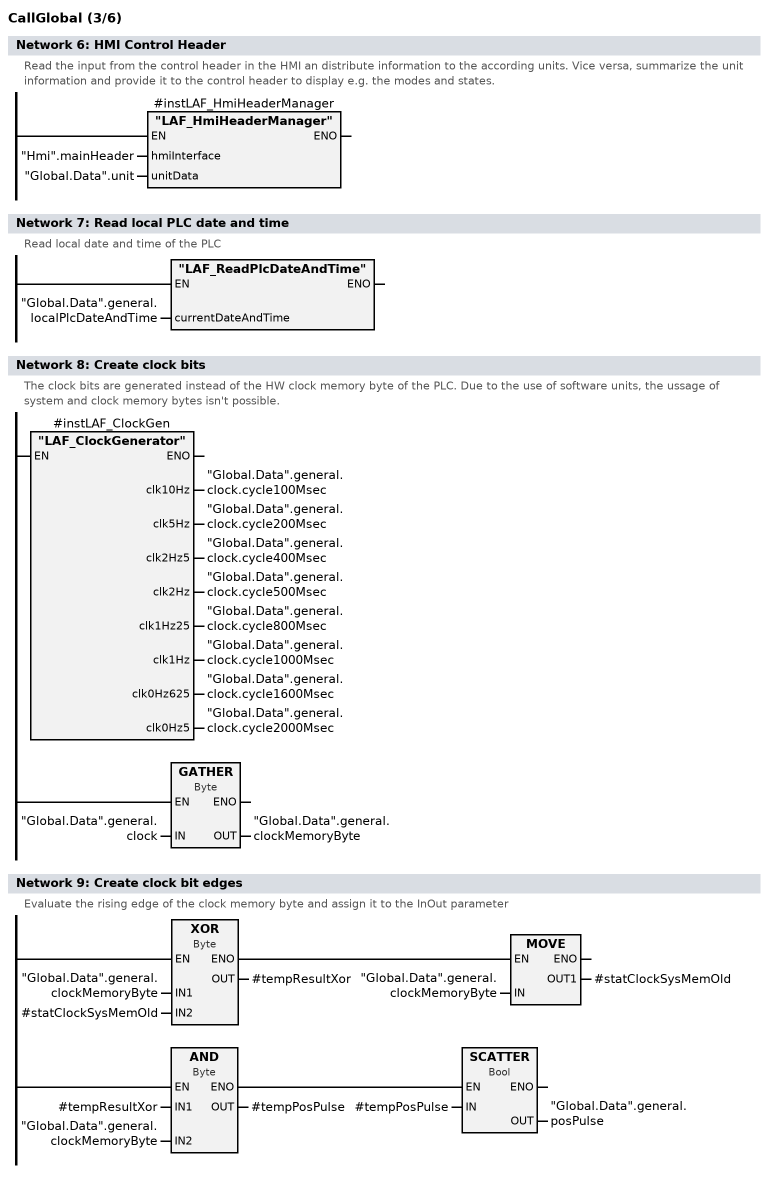
   RUNG wire#powerrail
      #instLAF_HmiHeaderManager(hmiInterface := "Hmi".mainHeader, unitData := "Global.Data".unit)
   END_RUNG
   // the same network as SCL:
   #instLAF_HmiHeaderManager(hmiInterface := "Hmi".mainHeader, unitData := "Global.Data".unit);   // "LAF_HmiHeaderManager"
END_REGION

REGION Network 7: Read local PLC date and time
   // Read local date and time of the PLC
   RUNG wire#powerrail
      "LAF_ReadPlcDateAndTime"(currentDateAndTime := "Global.Data".general.localPlcDateAndTime)
   END_RUNG
   // the same network as SCL:
   "LAF_ReadPlcDateAndTime"(currentDateAndTime := "Global.Data".general.localPlcDateAndTime);
END_REGION

REGION Network 8: Create clock bits
   // The clock bits are generated instead of the HW clock memory byte of the PLC. Due to the use of software units, the ussage of system and clock memory bytes isn't possible.
   RUNG wire#powerrail
      #instLAF_ClockGen(clk10Hz => "Global.Data".general.clock.cycle100Msec, clk5Hz => "Global.Data".general.clock.cycle200Msec, clk2Hz5 => "Global.Data".general.clock.cycle400Msec, clk2Hz => "Global.Data".general.clock.cycle500Msec, clk1Hz25 => "Global.Data".general.clock.cycle800Msec, clk1Hz => "Global.Data".general.clock.cycle1000Msec, clk0Hz625 => "Global.Data".general.clock.cycle1600Msec, clk0Hz5 => "Global.Data".general.clock.cycle2000Msec)
   END_RUNG
   RUNG wire#powerrail
      { S7_Templates := "[dest_type := Byte, src_type := Bool]" } GATHER(IN := "Global.Data".general.clock, OUT => "Global.Data".general.clockMemoryByte)
   END_RUNG
   // the same network as SCL:
   #instLAF_ClockGen(clk10Hz => "Global.Data".general.clock.cycle100Msec,   // "LAF_ClockGenerator"
                     clk5Hz => "Global.Data".general.clock.cycle200Msec,
                     clk2Hz5 => "Global.Data".general.clock.cycle400Msec,
                     clk2Hz => "Global.Data".general.clock.cycle500Msec,
                     clk1Hz25 => "Global.Data".general.clock.cycle800Msec,
                     clk1Hz => "Global.Data".general.clock.cycle1000Msec,
                     clk0Hz625 => "Global.Data".general.clock.cycle1600Msec,
                     clk0Hz5 => "Global.Data".general.clock.cycle2000Msec);
   GATHER(IN := "Global.Data".general.clock, OUT => "Global.Data".general.clockMemoryByte);
END_REGION

REGION Network 9: Create clock bit edges
   // Evaluate the rising edge of the clock memory byte and assign it to the InOut parameter
   #tempResultXor := "Global.Data".general.clockMemoryByte XOR #statClockSysMemOld;
   #statClockSysMemOld := "Global.Data".general.clockMemoryByte;
   #tempPosPulse := #tempResultXor AND "Global.Data".general.clockMemoryByte;
   SCATTER(IN := #tempPosPulse, OUT => "Global.Data".general.posPulse);
END_REGION

REGION Network 10: Time Synchronisation (NTP)
   // With the LSNTP_Server block, the NTP server will be enabled on S7 PLC, to wich the NTP client (e.g. Panel), can synchronize their data and time.
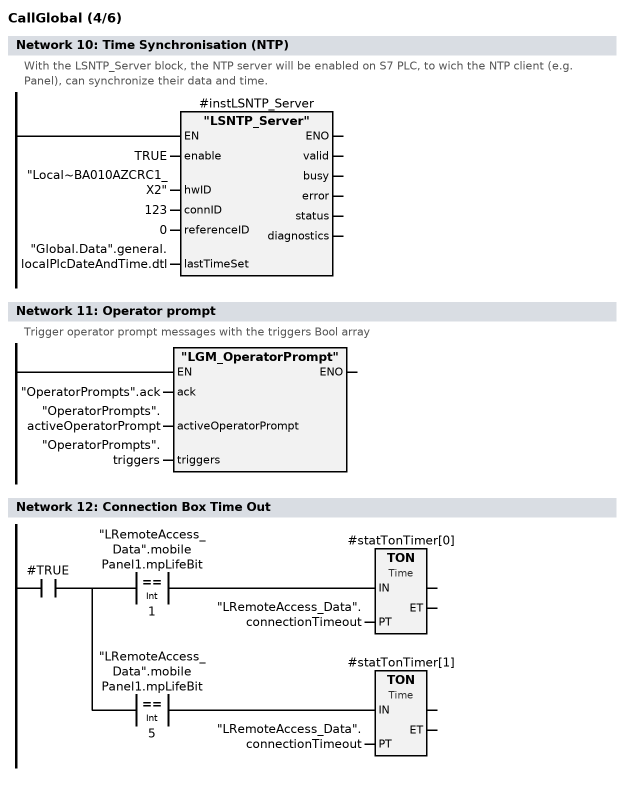
   RUNG wire#powerrail
      #instLSNTP_Server(enable := TRUE, hwID := "Local~BA010AZCRC1_X2", connID := 123, referenceID := 0, lastTimeSet := "Global.Data".general.localPlcDateAndTime.dtl, valid =>, busy =>, error =>, status =>, diagnostics =>)
   END_RUNG
   // the same network as SCL:
   #instLSNTP_Server(enable := TRUE,   // "LSNTP_Server"
                     hwID := "Local~BA010AZCRC1_X2",
                     connID := 123,
                     referenceID := 0,
                     lastTimeSet := "Global.Data".general.localPlcDateAndTime.dtl);
END_REGION

REGION Network 11: Operator prompt
   // Trigger operator prompt messages with the triggers Bool array
   RUNG wire#powerrail
      "LGM_OperatorPrompt"(ack := "OperatorPrompts".ack, activeOperatorPrompt := "OperatorPrompts".activeOperatorPrompt, triggers := "OperatorPrompts".triggers)
   END_RUNG
   // the same network as SCL:
   "LGM_OperatorPrompt"(ack := "OperatorPrompts".ack,
                        activeOperatorPrompt := "OperatorPrompts".activeOperatorPrompt,
                        triggers := "OperatorPrompts".triggers);
END_REGION

REGION Network 12: Connection Box Time Out
   RUNG wire#powerrail
      Contact( #TRUE )
      wire#w1
      { S7_Templates := "SrcType := Int" } EQ_Contact(in1 := "LRemoteAccess_Data".mobilePanel1.mpLifeBit, in2 := 1)
      { S7_Templates := "time_type := Time" } #statTonTimer[0].TON(pt := "LRemoteAccess_Data".connectionTimeout, et =>)
   END_RUNG
   RUNG wire#w1
      { S7_Templates := "SrcType := Int" } EQ_Contact(in1 := "LRemoteAccess_Data".mobilePanel1.mpLifeBit, in2 := 5)
      { S7_Templates := "time_type := Time" } #statTonTimer[1].TON(pt := "LRemoteAccess_Data".connectionTimeout, et =>)
   END_RUNG
   // the same network as SCL:
   #statTonTimer[0].TON(IN := #TRUE AND ("LRemoteAccess_Data".mobilePanel1.mpLifeBit = 1),
                        PT := "LRemoteAccess_Data".connectionTimeout);
   #statTonTimer[1].TON(IN := #TRUE AND ("LRemoteAccess_Data".mobilePanel1.mpLifeBit = 5),
                        PT := "LRemoteAccess_Data".connectionTimeout);
END_REGION

REGION Network 13: Connection box is connected
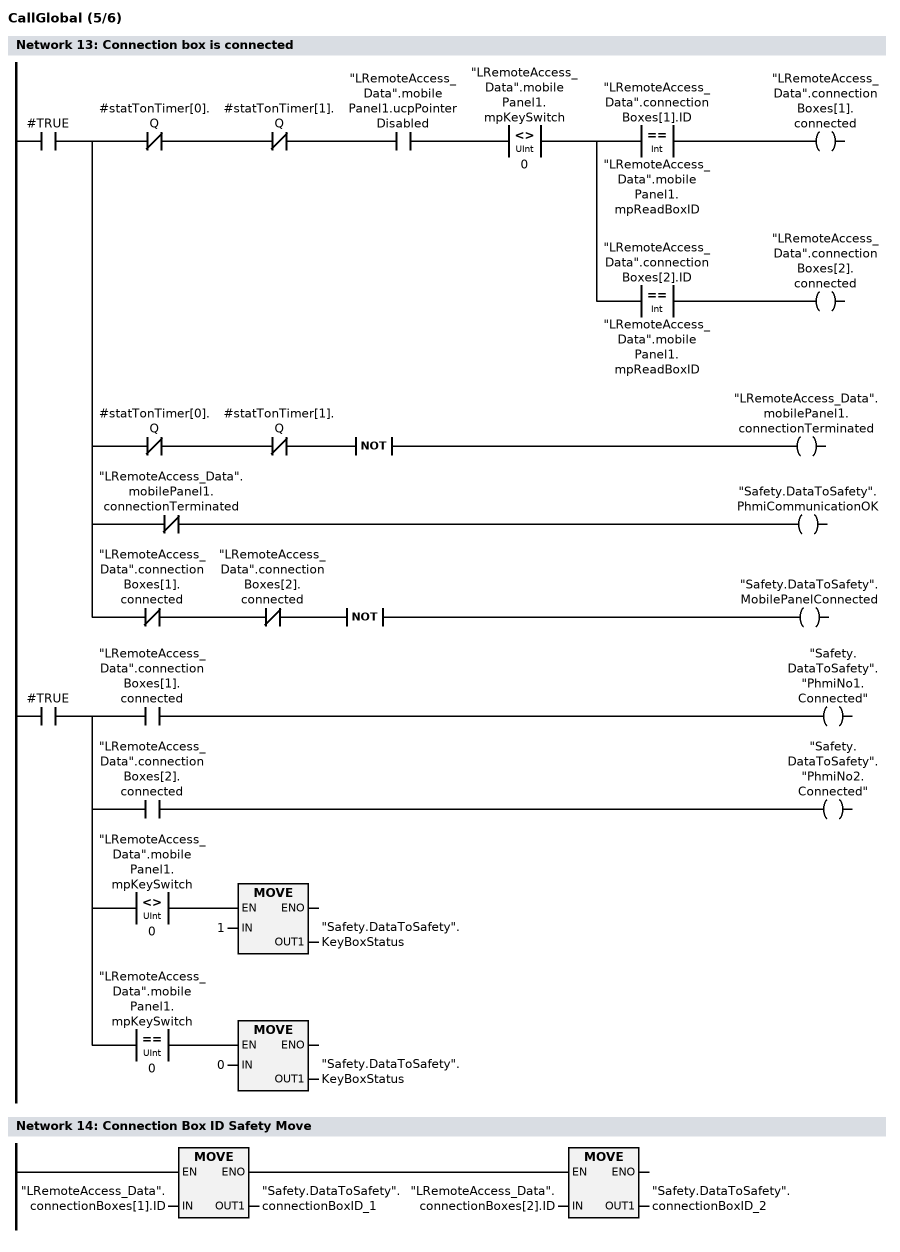
   RUNG wire#powerrail
      Contact( #TRUE )
      wire#w1
      I_Contact( #statTonTimer[0].Q )
      I_Contact( #statTonTimer[1].Q )
      Contact( "LRemoteAccess_Data".mobilePanel1.ucpPointerDisabled )
      { S7_Templates := "SrcType := UInt" } NE_Contact(in1 := "LRemoteAccess_Data".mobilePanel1.mpKeySwitch, in2 := 0)
      wire#w2
      { S7_Templates := "SrcType := Int" } EQ_Contact(in1 := "LRemoteAccess_Data".connectionBoxes[1].ID, in2 := "LRemoteAccess_Data".mobilePanel1.mpReadBoxID)
      Coil( "LRemoteAccess_Data".connectionBoxes[1].connected )
   END_RUNG
   RUNG wire#w2
      { S7_Templates := "SrcType := Int" } EQ_Contact(in1 := "LRemoteAccess_Data".connectionBoxes[2].ID, in2 := "LRemoteAccess_Data".mobilePanel1.mpReadBoxID)
      Coil( "LRemoteAccess_Data".connectionBoxes[2].connected )
   END_RUNG
   RUNG wire#w1
      I_Contact( #statTonTimer[0].Q )
      I_Contact( #statTonTimer[1].Q )
      Not()
      Coil( "LRemoteAccess_Data".mobilePanel1.connectionTerminated )
   END_RUNG
   RUNG wire#w1
      I_Contact( "LRemoteAccess_Data".mobilePanel1.connectionTerminated )
      Coil( "Safety.DataToSafety".PhmiCommunicationOK )
   END_RUNG
   RUNG wire#w1
      I_Contact( "LRemoteAccess_Data".connectionBoxes[1].connected )
      I_Contact( "LRemoteAccess_Data".connectionBoxes[2].connected )
      Not()
      Coil( "Safety.DataToSafety".MobilePanelConnected )
   END_RUNG
   RUNG wire#powerrail
      Contact( #TRUE )
      wire#w3
      Contact( "LRemoteAccess_Data".connectionBoxes[1].connected )
      Coil( "Safety.DataToSafety"."PhmiNo1.Connected" )
   END_RUNG
   RUNG wire#w3
      Contact( "LRemoteAccess_Data".connectionBoxes[2].connected )
      Coil( "Safety.DataToSafety"."PhmiNo2.Connected" )
   END_RUNG
   RUNG wire#w3
      { S7_Templates := "SrcType := UInt" } NE_Contact(in1 := "LRemoteAccess_Data".mobilePanel1.mpKeySwitch, in2 := 0)
      Move(in := 1, out1 => "Safety.DataToSafety".KeyBoxStatus)
   END_RUNG
   RUNG wire#w3
      { S7_Templates := "SrcType := UInt" } EQ_Contact(in1 := "LRemoteAccess_Data".mobilePanel1.mpKeySwitch, in2 := 0)
      Move(in := 0, out1 => "Safety.DataToSafety".KeyBoxStatus)
   END_RUNG
   // the same network as SCL:
   #_w1 := #TRUE AND NOT #statTonTimer[0].Q AND NOT #statTonTimer[1].Q AND "LRemoteAccess_Data".mobilePanel1.ucpPointerDisabled AND ("LRemoteAccess_Data".mobilePanel1.mpKeySwitch <> 0);
   "LRemoteAccess_Data".connectionBoxes[1].connected := #_w1 AND ("LRemoteAccess_Data".connectionBoxes[1].ID = "LRemoteAccess_Data".mobilePanel1.mpReadBoxID);
   "LRemoteAccess_Data".connectionBoxes[2].connected := #_w1 AND ("LRemoteAccess_Data".connectionBoxes[2].ID = "LRemoteAccess_Data".mobilePanel1.mpReadBoxID);
   "LRemoteAccess_Data".mobilePanel1.connectionTerminated := NOT (#TRUE AND NOT #statTonTimer[0].Q AND NOT #statTonTimer[1].Q);
   "Safety.DataToSafety".PhmiCommunicationOK := #TRUE AND NOT "LRemoteAccess_Data".mobilePanel1.connectionTerminated;
   "Safety.DataToSafety".MobilePanelConnected := NOT (#TRUE AND NOT "LRemoteAccess_Data".connectionBoxes[1].connected AND NOT "LRemoteAccess_Data".connectionBoxes[2].connected);
   "Safety.DataToSafety"."PhmiNo1.Connected" := #TRUE AND "LRemoteAccess_Data".connectionBoxes[1].connected;
   "Safety.DataToSafety"."PhmiNo2.Connected" := #TRUE AND "LRemoteAccess_Data".connectionBoxes[2].connected;
   IF #TRUE AND ("LRemoteAccess_Data".mobilePanel1.mpKeySwitch <> 0) THEN
       "Safety.DataToSafety".KeyBoxStatus := 1;
   END_IF;
   IF #TRUE AND ("LRemoteAccess_Data".mobilePanel1.mpKeySwitch = 0) THEN
       "Safety.DataToSafety".KeyBoxStatus := 0;
   END_IF;
END_REGION

REGION Network 14: Connection Box ID Safety Move
   RUNG wire#powerrail
      Move(in := "LRemoteAccess_Data".connectionBoxes[1].ID, out1 => "Safety.DataToSafety".connectionBoxID_1)
      Move(in := "LRemoteAccess_Data".connectionBoxes[2].ID, out1 => "Safety.DataToSafety".connectionBoxID_2)
   END_RUNG
   // the same network as SCL:
   "Safety.DataToSafety".connectionBoxID_1 := "LRemoteAccess_Data".connectionBoxes[1].ID;
   "Safety.DataToSafety".connectionBoxID_2 := "LRemoteAccess_Data".connectionBoxes[2].ID;
END_REGION

REGION Network 15: enable Control Interfaces
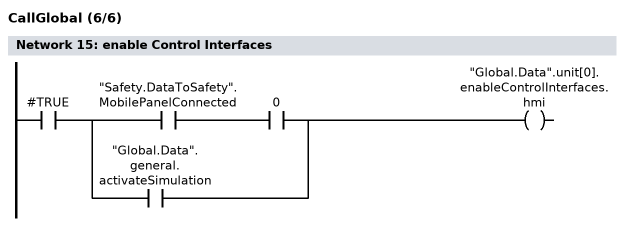
   RUNG wire#powerrail
      Contact( #TRUE )
      wire#w1
      Contact( "Safety.DataToSafety".MobilePanelConnected )
      Contact( 0 )
      wire#w2
      Coil( "Global.Data".unit[0].enableControlInterfaces.hmi )
   END_RUNG
   RUNG wire#w1
      Contact( "Global.Data".general.activateSimulation )
   END_RUNG wire#w2
   // the same network as SCL:
   "Global.Data".unit[0].enableControlInterfaces.hmi := #TRUE AND (("Safety.DataToSafety".MobilePanelConnected AND 0) OR "Global.Data".general.activateSimulation);
END_REGION
END_FUNCTION_BLOCK

FUNCTION "CallManualOperationLines_Unit1" : Void   // FC69, LAD
// stored: SetENOAutomatically false
   VAR_TEMP
      StatusEm : Array[0..7] of Struct
         Status : Array[0..45] of Word;
      END_STRUCT;
      errorIDEm : Array[0..7] of Struct
         errorID : Array[0..45] of Word;
      END_STRUCT;
      disableUnit1 : Bool;
      TempAxisCommands : "LBC_typeAxis64PosManualCommands";
      TempAxisMonitoring : "LBC_typeAxis64PosProcessValues";
      TempSoftCam : Array[0..8] of "LER_typeSoftCamParameter";
   END_VAR
   VAR CONSTANT
      MECHANIC_NAME_ENABLE : Bool;
   END_VAR
BEGIN

REGION Network 1: Unit 1 Enable Manual Operation
   // Condition to disable manual operation lines in Unit 1
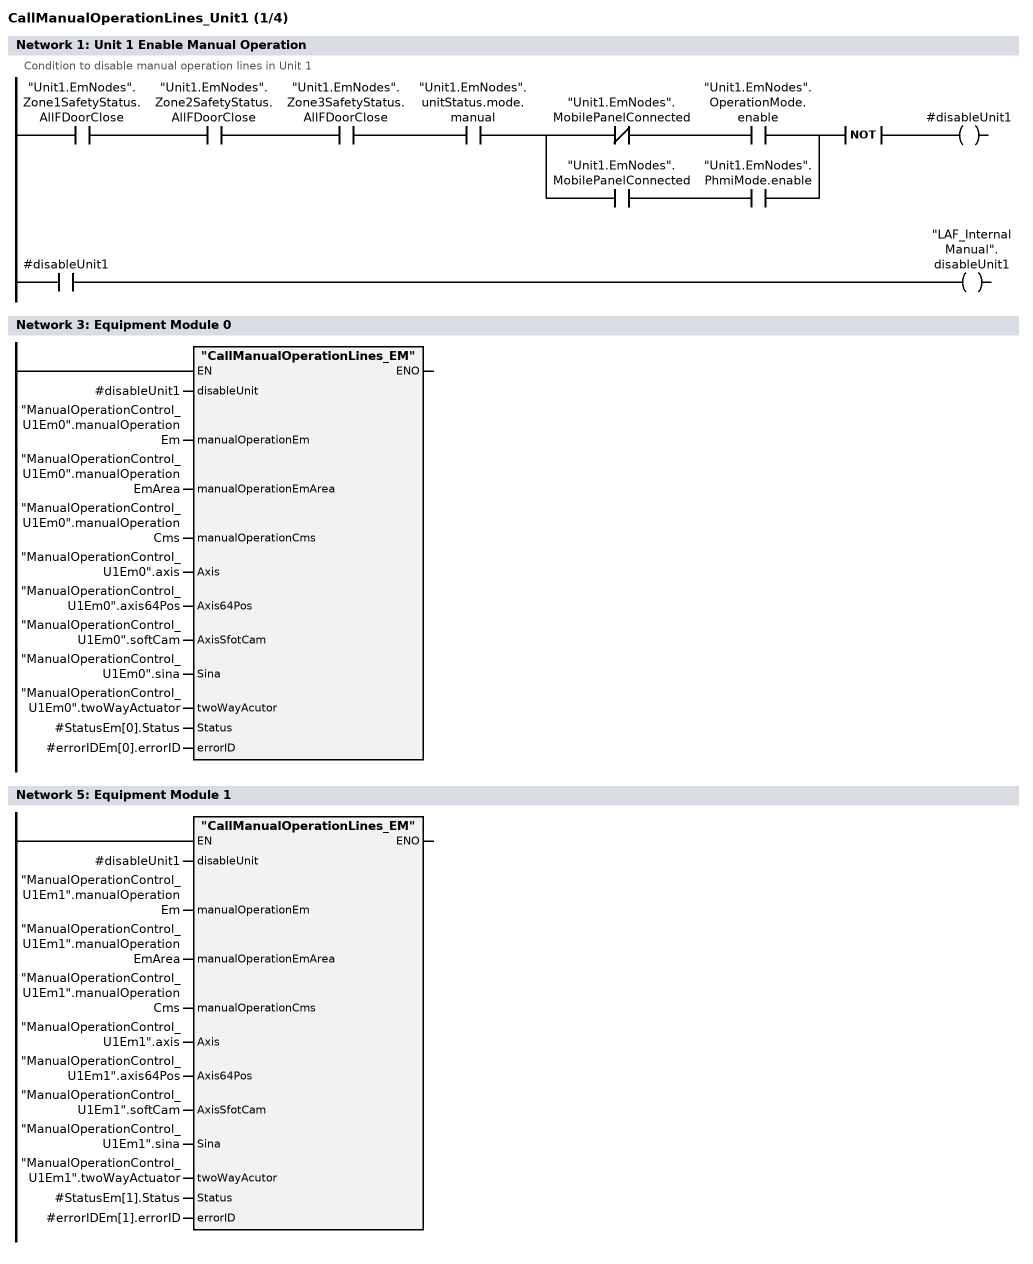
   RUNG wire#powerrail
      Contact( "Unit1.EmNodes".Zone1SafetyStatus.AllFDoorClose )
      Contact( "Unit1.EmNodes".Zone2SafetyStatus.AllFDoorClose )
      Contact( "Unit1.EmNodes".Zone3SafetyStatus.AllFDoorClose )
      Contact( "Unit1.EmNodes".unitStatus.mode.manual )
      wire#w1
      I_Contact( "Unit1.EmNodes".MobilePanelConnected )
      Contact( "Unit1.EmNodes".OperationMode.enable )
      wire#w2
      Not()
      Coil( #disableUnit1 )
   END_RUNG
   RUNG wire#w1
      Contact( "Unit1.EmNodes".MobilePanelConnected )
      Contact( "Unit1.EmNodes".PhmiMode.enable )
   END_RUNG wire#w2
   RUNG wire#powerrail
      Contact( #disableUnit1 )
      Coil( "LAF_InternalManual".disableUnit1 )
   END_RUNG
   // the same network as SCL:
   #disableUnit1 := NOT ("Unit1.EmNodes".Zone1SafetyStatus.AllFDoorClose AND "Unit1.EmNodes".Zone2SafetyStatus.AllFDoorClose AND "Unit1.EmNodes".Zone3SafetyStatus.AllFDoorClose AND "Unit1.EmNodes".unitStatus.mode.manual AND ((NOT "Unit1.EmNodes".MobilePanelConnected AND "Unit1.EmNodes".OperationMode.enable) OR ("Unit1.EmNodes".MobilePanelConnected AND "Unit1.EmNodes".PhmiMode.enable)));
   "LAF_InternalManual".disableUnit1 := #disableUnit1;
END_REGION

REGION Network 2 (SCL): Equipment Module 0 Cms Mapping
   REGION Input Mapping
       // Axis
       "ManualOperationControl_U1Em0".axis[1].monitoring := "Unit1.Em0.HmiInterface".cmUnWinderAxisB.monitoring;

       // TwoWayActuator
       "ManualOperationControl_U1Em0".twoWayActuator[1].monitoring := "Unit1.Em0.HmiInterface".cmAirShaftOnOff.monitoring;
       "ManualOperationControl_U1Em0".twoWayActuator[2].monitoring := "Unit1.Em0.HmiInterface".cmExpelFwdBwd.monitoring;
   END_REGION


   REGION Output Mapping
       // Axis
       "CallManualOperationLines_ServoCommands"(ManualOperationControl := "ManualOperationControl_U1Em0".axis[1].commands,
                                                HmiInterface => "Unit1.Em0.HmiInterface".cmUnWinderAxisB.commands);

       // TwoWayActuator
       "Unit1.Em0.HmiInterface".cmAirShaftOnOff.commands := "ManualOperationControl_U1Em0".twoWayActuator[1].commands;
       "Unit1.Em0.HmiInterface".cmExpelFwdBwd.commands := "ManualOperationControl_U1Em0".twoWayActuator[2].commands;
   END_REGION
END_REGION

REGION Network 3: Equipment Module 0
   RUNG wire#powerrail
      "CallManualOperationLines_EM"(disableUnit := #disableUnit1, manualOperationEm := "ManualOperationControl_U1Em0".manualOperationEm, manualOperationEmArea := "ManualOperationControl_U1Em0".manualOperationEmArea, manualOperationCms := "ManualOperationControl_U1Em0".manualOperationCms, Axis := "ManualOperationControl_U1Em0".axis, Axis64Pos := "ManualOperationControl_U1Em0".axis64Pos, AxisSfotCam := "ManualOperationControl_U1Em0".softCam, Sina := "ManualOperationControl_U1Em0".sina, twoWayAcutor := "ManualOperationControl_U1Em0".twoWayActuator, Status := #StatusEm[0].Status, errorID := #errorIDEm[0].errorID)
   END_RUNG
   // the same network as SCL:
   "CallManualOperationLines_EM"(disableUnit := #disableUnit1,
                           manualOperationEm := "ManualOperationControl_U1Em0".manualOperationEm,
                           manualOperationEmArea := "ManualOperationControl_U1Em0".manualOperationEmArea,
                           manualOperationCms := "ManualOperationControl_U1Em0".manualOperationCms,
                           Axis := "ManualOperationControl_U1Em0".axis,
                           Axis64Pos := "ManualOperationControl_U1Em0".axis64Pos,
                           AxisSfotCam := "ManualOperationControl_U1Em0".softCam,
                           Sina := "ManualOperationControl_U1Em0".sina,
                           twoWayAcutor := "ManualOperationControl_U1Em0".twoWayActuator,
                           Status := #StatusEm[0].Status,
                           errorID := #errorIDEm[0].errorID);
END_REGION

REGION Network 4 (SCL): Equipment Module 1 Cms Mapping
   REGION Input Mapping
       // Axis
       "ManualOperationControl_U1Em1".axis[1].monitoring := "Unit1.Em1.HmiInterface".cmUnWinderAxisB.monitoring;

       // TwoWayActuator
       "ManualOperationControl_U1Em1".twoWayActuator[1].monitoring := "Unit1.Em1.HmiInterface".cmAirShaftOnOff.monitoring;
       "ManualOperationControl_U1Em1".twoWayActuator[2].monitoring := "Unit1.Em1.HmiInterface".cmExpelFwdBwd.monitoring;
   END_REGION


   REGION Output Mapping
       // Axis
       "CallManualOperationLines_ServoCommands"(ManualOperationControl := "ManualOperationControl_U1Em1".axis[1].commands,
                                                HmiInterface => "Unit1.Em1.HmiInterface".cmUnWinderAxisB.commands);

       // TwoWayActuator
       "Unit1.Em1.HmiInterface".cmAirShaftOnOff.commands := "ManualOperationControl_U1Em1".twoWayActuator[1].commands;
       "Unit1.Em1.HmiInterface".cmExpelFwdBwd.commands := "ManualOperationControl_U1Em1".twoWayActuator[2].commands;
   END_REGION
END_REGION

REGION Network 5: Equipment Module 1
   RUNG wire#powerrail
      "CallManualOperationLines_EM"(disableUnit := #disableUnit1, manualOperationEm := "ManualOperationControl_U1Em1".manualOperationEm, manualOperationEmArea := "ManualOperationControl_U1Em1".manualOperationEmArea, manualOperationCms := "ManualOperationControl_U1Em1".manualOperationCms, Axis := "ManualOperationControl_U1Em1".axis, Axis64Pos := "ManualOperationControl_U1Em1".axis64Pos, AxisSfotCam := "ManualOperationControl_U1Em1".softCam, Sina := "ManualOperationControl_U1Em1".sina, twoWayAcutor := "ManualOperationControl_U1Em1".twoWayActuator, Status := #StatusEm[1].Status, errorID := #errorIDEm[1].errorID)
   END_RUNG
   // the same network as SCL:
   "CallManualOperationLines_EM"(disableUnit := #disableUnit1,
                           manualOperationEm := "ManualOperationControl_U1Em1".manualOperationEm,
                           manualOperationEmArea := "ManualOperationControl_U1Em1".manualOperationEmArea,
                           manualOperationCms := "ManualOperationControl_U1Em1".manualOperationCms,
                           Axis := "ManualOperationControl_U1Em1".axis,
                           Axis64Pos := "ManualOperationControl_U1Em1".axis64Pos,
                           AxisSfotCam := "ManualOperationControl_U1Em1".softCam,
                           Sina := "ManualOperationControl_U1Em1".sina,
                           twoWayAcutor := "ManualOperationControl_U1Em1".twoWayActuator,
                           Status := #StatusEm[1].Status,
                           errorID := #errorIDEm[1].errorID);
END_REGION

REGION Network 6 (SCL): Equipment Module 2 Cms Mapping
   REGION Input Mapping
       // TwoWayActuator
       "ManualOperationControl_U1Em2".twoWayActuator[1].monitoring := "Unit1.Em2.HmiInterface".cmElectrodeFixRightTopFwdBwd.monitoring;
       "ManualOperationControl_U1Em2".twoWayActuator[2].monitoring := "Unit1.Em2.HmiInterface".cmElectrodeFixRightBottomFwdBwd.monitoring;
       "ManualOperationControl_U1Em2".twoWayActuator[3].monitoring := "Unit1.Em2.HmiInterface".cmElectrodeFixLeftTopFwdBwd.monitoring;
       "ManualOperationControl_U1Em2".twoWayActuator[4].monitoring := "Unit1.Em2.HmiInterface".cmElectrodeFixLeftBottomFwdBwd.monitoring;
       "ManualOperationControl_U1Em2".twoWayActuator[5].monitoring := "Unit1.Em2.HmiInterface".cmElectrodeFixLeftTopUpDown.monitoring;
       "ManualOperationControl_U1Em2".twoWayActuator[6].monitoring := "Unit1.Em2.HmiInterface".cmElectrodeFixLeftBottomUpDown.monitoring;
       "ManualOperationControl_U1Em2".twoWayActuator[7].monitoring := "Unit1.Em2.HmiInterface".cmUwSemiSplicerVacuumRightTopOnOff.monitoring;
       "ManualOperationControl_U1Em2".twoWayActuator[8].monitoring := "Unit1.Em2.HmiInterface".cmUwSemiSplicerVacuumRightBottomOnOff.monitoring;
       "ManualOperationControl_U1Em2".twoWayActuator[9].monitoring := "Unit1.Em2.HmiInterface".cmUwSemiSplicerVacuumLeftTopOnOff.monitoring;
       "ManualOperationControl_U1Em2".twoWayActuator[10].monitoring := "Unit1.Em2.HmiInterface".cmUwSemiSplicerVacuumLeftBottomOnOff.monitoring;
       "ManualOperationControl_U1Em2".twoWayActuator[11].monitoring := "Unit1.Em2.HmiInterface".cmElectrodeCutterFwdBwd.monitoring;
       "ManualOperationControl_U1Em2".twoWayActuator[12].monitoring := "Unit1.Em2.HmiInterface".cmSplicingLeftModuleMoverFwdBwd.monitoring;
       "ManualOperationControl_U1Em2".twoWayActuator[13].monitoring := "Unit1.Em2.HmiInterface".cmSplicingRightModuleMoverFwdBwd.monitoring;
       "ManualOperationControl_U1Em2".twoWayActuator[14].monitoring := "Unit1.Em2.HmiInterface".cmElectrodeLeftHolderMoverFwdBwd.monitoring;
       "ManualOperationControl_U1Em2".twoWayActuator[15].monitoring := "Unit1.Em2.HmiInterface".cmElectrodeRightHolderMoverFwdBwd.monitoring;
       "ManualOperationControl_U1Em2".twoWayActuator[16].monitoring := "Unit1.Em2.HmiInterface".cmTapeLoadingTurnCwCcw.monitoring;
       "ManualOperationControl_U1Em2".twoWayActuator[17].monitoring := "Unit1.Em2.HmiInterface".cmTapeAttachUnitFwdBwd.monitoring;
       "ManualOperationControl_U1Em2".twoWayActuator[18].monitoring := "Unit1.Em2.HmiInterface".cmTapeVacuumOnOff.monitoring;
       "ManualOperationControl_U1Em2".twoWayActuator[19].monitoring := "Unit1.Em2.HmiInterface".cmStopperFwdBwd.monitoring;
       "ManualOperationControl_U1Em2".twoWayActuator[20].monitoring := "Unit1.Em2.HmiInterface".cmSupportUnitTransferFwdBwd.monitoring;
       "ManualOperationControl_U1Em2".twoWayActuator[21].monitoring := "Unit1.Em2.HmiInterface".cmSupportUnitShaftUpDown.monitoring;
       "ManualOperationControl_U1Em2".twoWayActuator[22].monitoring := "Unit1.Em2.HmiInterface".cmFrameCoverFwdBwd.monitoring;
   END_REGION


   REGION Output Mapping
       // TwoWayActuator
       "Unit1.Em2.HmiInterface".cmElectrodeFixRightTopFwdBwd.commands := "ManualOperationControl_U1Em2".twoWayActuator[1].commands;
       "Unit1.Em2.HmiInterface".cmElectrodeFixRightBottomFwdBwd.commands := "ManualOperationControl_U1Em2".twoWayActuator[2].commands;
       "Unit1.Em2.HmiInterface".cmElectrodeFixLeftTopFwdBwd.commands := "ManualOperationControl_U1Em2".twoWayActuator[3].commands;
       "Unit1.Em2.HmiInterface".cmElectrodeFixLeftBottomFwdBwd.commands := "ManualOperationControl_U1Em2".twoWayActuator[4].commands;
       "Unit1.Em2.HmiInterface".cmElectrodeFixLeftTopUpDown.commands := "ManualOperationControl_U1Em2".twoWayActuator[5].commands;
       "Unit1.Em2.HmiInterface".cmElectrodeFixLeftBottomUpDown.commands := "ManualOperationControl_U1Em2".twoWayActuator[6].commands;
       "Unit1.Em2.HmiInterface".cmUwSemiSplicerVacuumRightTopOnOff.commands := "ManualOperationControl_U1Em2".twoWayActuator[7].commands;
       "Unit1.Em2.HmiInterface".cmUwSemiSplicerVacuumRightBottomOnOff.commands := "ManualOperationControl_U1Em2".twoWayActuator[8].commands;
       "Unit1.Em2.HmiInterface".cmUwSemiSplicerVacuumLeftTopOnOff.commands := "ManualOperationControl_U1Em2".twoWayActuator[9].commands;
       "Unit1.Em2.HmiInterface".cmUwSemiSplicerVacuumLeftBottomOnOff.commands := "ManualOperationControl_U1Em2".twoWayActuator[10].commands;
       "Unit1.Em2.HmiInterface".cmElectrodeCutterFwdBwd.commands := "ManualOperationControl_U1Em2".twoWayActuator[11].commands;
       "Unit1.Em2.HmiInterface".cmSplicingLeftModuleMoverFwdBwd.commands := "ManualOperationControl_U1Em2".twoWayActuator[12].commands;
       "Unit1.Em2.HmiInterface".cmSplicingRightModuleMoverFwdBwd.commands := "ManualOperationControl_U1Em2".twoWayActuator[13].commands;
       "Unit1.Em2.HmiInterface".cmElectrodeLeftHolderMoverFwdBwd.commands := "ManualOperationControl_U1Em2".twoWayActuator[14].commands;
       "Unit1.Em2.HmiInterface".cmElectrodeRightHolderMoverFwdBwd.commands := "ManualOperationControl_U1Em2".twoWayActuator[15].commands;
       "Unit1.Em2.HmiInterface".cmTapeLoadingTurnCwCcw.commands := "ManualOperationControl_U1Em2".twoWayActuator[16].commands;
       "Unit1.Em2.HmiInterface".cmTapeAttachUnitFwdBwd.commands := "ManualOperationControl_U1Em2".twoWayActuator[17].commands;
       "Unit1.Em2.HmiInterface".cmTapeVacuumOnOff.commands := "ManualOperationControl_U1Em2".twoWayActuator[18].commands;
       "Unit1.Em2.HmiInterface".cmStopperFwdBwd.commands := "ManualOperationControl_U1Em2".twoWayActuator[19].commands;
       "Unit1.Em2.HmiInterface".cmSupportUnitTransferFwdBwd.commands := "ManualOperationControl_U1Em2".twoWayActuator[20].commands;
       "Unit1.Em2.HmiInterface".cmSupportUnitShaftUpDown.commands := "ManualOperationControl_U1Em2".twoWayActuator[21].commands;
       "Unit1.Em2.HmiInterface".cmFrameCoverFwdBwd.commands := "ManualOperationControl_U1Em2".twoWayActuator[22].commands;
   END_REGION
END_REGION

REGION Network 7: Equipment Module 2
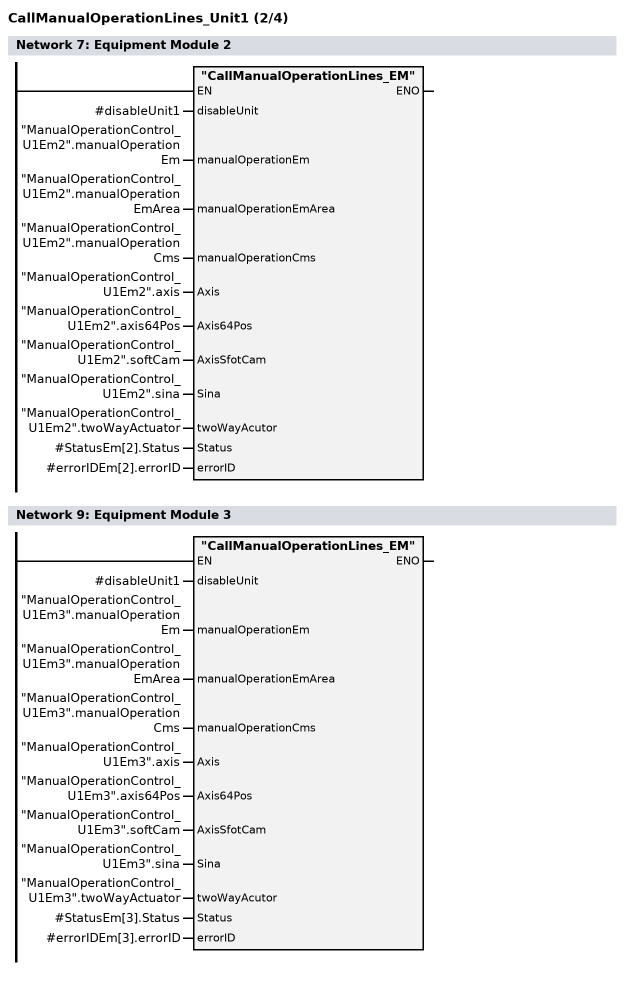
   RUNG wire#powerrail
      "CallManualOperationLines_EM"(disableUnit := #disableUnit1, manualOperationEm := "ManualOperationControl_U1Em2".manualOperationEm, manualOperationEmArea := "ManualOperationControl_U1Em2".manualOperationEmArea, manualOperationCms := "ManualOperationControl_U1Em2".manualOperationCms, Axis := "ManualOperationControl_U1Em2".axis, Axis64Pos := "ManualOperationControl_U1Em2".axis64Pos, AxisSfotCam := "ManualOperationControl_U1Em2".softCam, Sina := "ManualOperationControl_U1Em2".sina, twoWayAcutor := "ManualOperationControl_U1Em2".twoWayActuator, Status := #StatusEm[2].Status, errorID := #errorIDEm[2].errorID)
   END_RUNG
   // the same network as SCL:
   "CallManualOperationLines_EM"(disableUnit := #disableUnit1,
                           manualOperationEm := "ManualOperationControl_U1Em2".manualOperationEm,
                           manualOperationEmArea := "ManualOperationControl_U1Em2".manualOperationEmArea,
                           manualOperationCms := "ManualOperationControl_U1Em2".manualOperationCms,
                           Axis := "ManualOperationControl_U1Em2".axis,
                           Axis64Pos := "ManualOperationControl_U1Em2".axis64Pos,
                           AxisSfotCam := "ManualOperationControl_U1Em2".softCam,
                           Sina := "ManualOperationControl_U1Em2".sina,
                           twoWayAcutor := "ManualOperationControl_U1Em2".twoWayActuator,
                           Status := #StatusEm[2].Status,
                           errorID := #errorIDEm[2].errorID);
END_REGION

REGION Network 8 (SCL): Equipment Module 3 Cms Mapping
   REGION Input Mapping
       // TwoWayActuator
       "ManualOperationControl_U1Em3".twoWayActuator[1].monitoring := "Unit1.Em3.HmiInterface".cmDancerRegulatorOnOff.monitoring;
   END_REGION


   REGION Output Mapping
       // TwoWayActuator
       "Unit1.Em3.HmiInterface".cmDancerRegulatorOnOff.commands := "ManualOperationControl_U1Em3".twoWayActuator[1].commands;
   END_REGION
END_REGION

REGION Network 9: Equipment Module 3
   RUNG wire#powerrail
      "CallManualOperationLines_EM"(disableUnit := #disableUnit1, manualOperationEm := "ManualOperationControl_U1Em3".manualOperationEm, manualOperationEmArea := "ManualOperationControl_U1Em3".manualOperationEmArea, manualOperationCms := "ManualOperationControl_U1Em3".manualOperationCms, Axis := "ManualOperationControl_U1Em3".axis, Axis64Pos := "ManualOperationControl_U1Em3".axis64Pos, AxisSfotCam := "ManualOperationControl_U1Em3".softCam, Sina := "ManualOperationControl_U1Em3".sina, twoWayAcutor := "ManualOperationControl_U1Em3".twoWayActuator, Status := #StatusEm[3].Status, errorID := #errorIDEm[3].errorID)
   END_RUNG
   // the same network as SCL:
   "CallManualOperationLines_EM"(disableUnit := #disableUnit1,
                           manualOperationEm := "ManualOperationControl_U1Em3".manualOperationEm,
                           manualOperationEmArea := "ManualOperationControl_U1Em3".manualOperationEmArea,
                           manualOperationCms := "ManualOperationControl_U1Em3".manualOperationCms,
                           Axis := "ManualOperationControl_U1Em3".axis,
                           Axis64Pos := "ManualOperationControl_U1Em3".axis64Pos,
                           AxisSfotCam := "ManualOperationControl_U1Em3".softCam,
                           Sina := "ManualOperationControl_U1Em3".sina,
                           twoWayAcutor := "ManualOperationControl_U1Em3".twoWayActuator,
                           Status := #StatusEm[3].Status,
                           errorID := #errorIDEm[3].errorID);
END_REGION

REGION Network 10 (SCL): Equipment Module 4 Cms Mapping
   REGION Input Mapping
       // Axis
       "ManualOperationControl_U1Em4".axis[1].monitoring := "Unit1.Em4.HmiInterface".cmCompensatorAxisZ.monitoring;
       "ManualOperationControl_U1Em4".axis[2].monitoring := "Unit1.Em4.HmiInterface".cmFeedingRollAxisB.monitoring;
       "ManualOperationControl_U1Em4".axis[3].monitoring := "Unit1.Em4.HmiInterface".cmElectrodeCutterAxisZ.monitoring;
       "ManualOperationControl_U1Em4".axis64Pos[1].monitoring := "Unit1.Em4.HmiInterface".cmPositionMovingAxisX.monitoring;

       // SoftCam
       "ManualOperationControl_U1Em4".softCam[1] := "Unit1.Em4.HmiInterface".cm.softcam.positionMoving;

       // TwoWayActuator
       "ManualOperationControl_U1Em4".twoWayActuator[1].monitoring := "Unit1.Em4.HmiInterface".cmFeederCylinderUpDown.monitoring;
   END_REGION


   REGION Output Mapping
       // Axis
       "CallManualOperationLines_ServoCommands"(ManualOperationControl := "ManualOperationControl_U1Em4".axis[1].commands,
                                                HmiInterface => "Unit1.Em4.HmiInterface".cmCompensatorAxisZ.commands);
       "CallManualOperationLines_ServoCommands"(ManualOperationControl := "ManualOperationControl_U1Em4".axis[2].commands,
                                                HmiInterface => "Unit1.Em4.HmiInterface".cmFeedingRollAxisB.commands);
       "CallManualOperationLines_ServoCommands"(ManualOperationControl := "ManualOperationControl_U1Em4".axis[3].commands,
                                                HmiInterface => "Unit1.Em4.HmiInterface".cmElectrodeCutterAxisZ.commands);
       "CallManualOperationLines_ServoPos64Commands"(ManualOperationControl := "ManualOperationControl_U1Em4".axis64Pos[1].commands,
                                                     HmiInterface => "Unit1.Em4.HmiInterface".cmPositionMovingAxisX.commands);

       // TwoWayActuator
       "Unit1.Em4.HmiInterface".cmFeederCylinderUpDown.commands := "ManualOperationControl_U1Em4".twoWayActuator[1].commands;
   END_REGION
END_REGION

REGION Network 11: Equipment Module 4
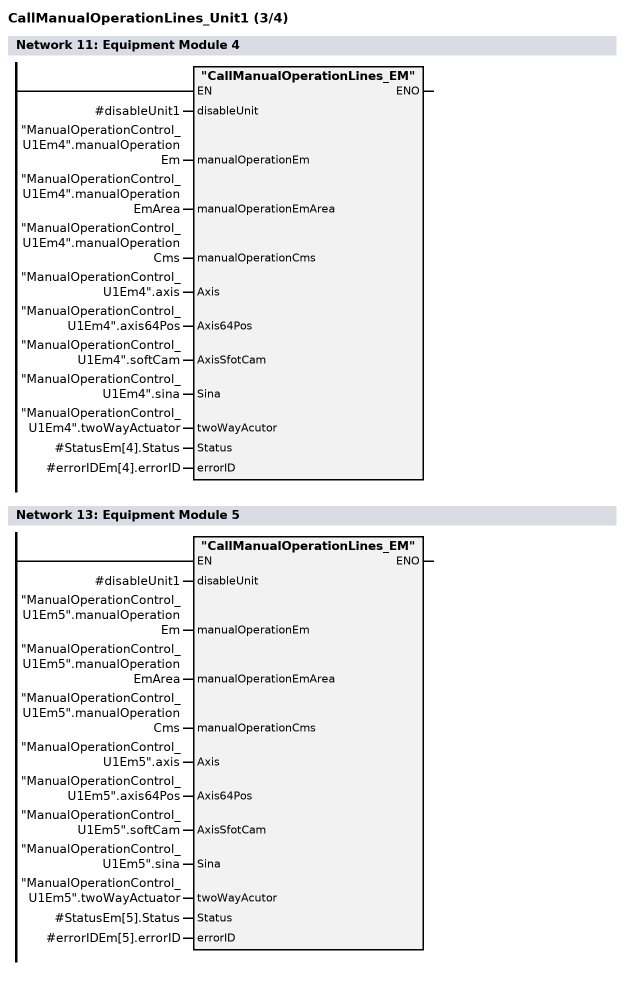
   RUNG wire#powerrail
      "CallManualOperationLines_EM"(disableUnit := #disableUnit1, manualOperationEm := "ManualOperationControl_U1Em4".manualOperationEm, manualOperationEmArea := "ManualOperationControl_U1Em4".manualOperationEmArea, manualOperationCms := "ManualOperationControl_U1Em4".manualOperationCms, Axis := "ManualOperationControl_U1Em4".axis, Axis64Pos := "ManualOperationControl_U1Em4".axis64Pos, AxisSfotCam := "ManualOperationControl_U1Em4".softCam, Sina := "ManualOperationControl_U1Em4".sina, twoWayAcutor := "ManualOperationControl_U1Em4".twoWayActuator, Status := #StatusEm[4].Status, errorID := #errorIDEm[4].errorID)
   END_RUNG
   // the same network as SCL:
   "CallManualOperationLines_EM"(disableUnit := #disableUnit1,
                           manualOperationEm := "ManualOperationControl_U1Em4".manualOperationEm,
                           manualOperationEmArea := "ManualOperationControl_U1Em4".manualOperationEmArea,
                           manualOperationCms := "ManualOperationControl_U1Em4".manualOperationCms,
                           Axis := "ManualOperationControl_U1Em4".axis,
                           Axis64Pos := "ManualOperationControl_U1Em4".axis64Pos,
                           AxisSfotCam := "ManualOperationControl_U1Em4".softCam,
                           Sina := "ManualOperationControl_U1Em4".sina,
                           twoWayAcutor := "ManualOperationControl_U1Em4".twoWayActuator,
                           Status := #StatusEm[4].Status,
                           errorID := #errorIDEm[4].errorID);
END_REGION

REGION Network 12 (SCL): Equipment Module 5 Cms Mapping
   REGION Input Mapping
       // Axis
       "ManualOperationControl_U1Em5".axis64Pos[1].monitoring := "Unit1.Em5.HmiInterface".cmNgAndManualInputAxisY.monitoring;
       "ManualOperationControl_U1Em5".axis64Pos[2].monitoring := "Unit1.Em5.HmiInterface".cmMagazineAxisZ.monitoring;

       // SoftCam
       "ManualOperationControl_U1Em5".softCam[1] := "Unit1.Em5.HmiInterface".cm.softcam.ngAndManualInput;
       "ManualOperationControl_U1Em5".softCam[2] := "Unit1.Em5.HmiInterface".cm.softcam.magazine;

       // TwoWayActuator
       "ManualOperationControl_U1Em5".twoWayActuator[1].monitoring := "Unit1.Em5.HmiInterface".cmNgAndManualInputCylinderUpDown.monitoring;
       "ManualOperationControl_U1Em5".twoWayActuator[2].monitoring := "Unit1.Em5.HmiInterface".cmNgAndManualInputVacuum1OnOff.monitoring;
       "ManualOperationControl_U1Em5".twoWayActuator[3].monitoring := "Unit1.Em5.HmiInterface".cmNgAndManualInputVacuum2OnOff.monitoring;
       "ManualOperationControl_U1Em5".twoWayActuator[4].monitoring := "Unit1.Em5.HmiInterface".cmNgAndManualInputVibrator1OnOff.monitoring;
       "ManualOperationControl_U1Em5".twoWayActuator[5].monitoring := "Unit1.Em5.HmiInterface".cmNgAndManualInputVibrator2OnOff.monitoring;
       "ManualOperationControl_U1Em5".twoWayActuator[6].monitoring := "Unit1.Em5.HmiInterface".cmMagazineLockCylinderUpDown.monitoring;
   END_REGION


   REGION Output Mapping
       // Axis
       "CallManualOperationLines_ServoPos64Commands"(ManualOperationControl := "ManualOperationControl_U1Em5".axis64Pos[1].commands,
                                                     HmiInterface => "Unit1.Em5.HmiInterface".cmNgAndManualInputAxisY.commands);
       "CallManualOperationLines_ServoPos64Commands"(ManualOperationControl := "ManualOperationControl_U1Em5".axis64Pos[2].commands,
                                                     HmiInterface => "Unit1.Em5.HmiInterface".cmMagazineAxisZ.commands);

       // TwoWayActuator
       "Unit1.Em5.HmiInterface".cmNgAndManualInputCylinderUpDown.commands := "ManualOperationControl_U1Em5".twoWayActuator[1].commands;
       "Unit1.Em5.HmiInterface".cmNgAndManualInputVacuum1OnOff.commands := "ManualOperationControl_U1Em5".twoWayActuator[2].commands;
       "Unit1.Em5.HmiInterface".cmNgAndManualInputVacuum2OnOff.commands := "ManualOperationControl_U1Em5".twoWayActuator[3].commands;
       "Unit1.Em5.HmiInterface".cmNgAndManualInputVibrator1OnOff.commands := "ManualOperationControl_U1Em5".twoWayActuator[4].commands;
       "Unit1.Em5.HmiInterface".cmNgAndManualInputVibrator2OnOff.commands := "ManualOperationControl_U1Em5".twoWayActuator[5].commands;
       "Unit1.Em5.HmiInterface".cmMagazineLockCylinderUpDown.commands := "ManualOperationControl_U1Em5".twoWayActuator[6].commands;
   END_REGION
END_REGION

REGION Network 13: Equipment Module 5
   RUNG wire#powerrail
      "CallManualOperationLines_EM"(disableUnit := #disableUnit1, manualOperationEm := "ManualOperationControl_U1Em5".manualOperationEm, manualOperationEmArea := "ManualOperationControl_U1Em5".manualOperationEmArea, manualOperationCms := "ManualOperationControl_U1Em5".manualOperationCms, Axis := "ManualOperationControl_U1Em5".axis, Axis64Pos := "ManualOperationControl_U1Em5".axis64Pos, AxisSfotCam := "ManualOperationControl_U1Em5".softCam, Sina := "ManualOperationControl_U1Em5".sina, twoWayAcutor := "ManualOperationControl_U1Em5".twoWayActuator, Status := #StatusEm[5].Status, errorID := #errorIDEm[5].errorID)
   END_RUNG
   // the same network as SCL:
   "CallManualOperationLines_EM"(disableUnit := #disableUnit1,
                           manualOperationEm := "ManualOperationControl_U1Em5".manualOperationEm,
                           manualOperationEmArea := "ManualOperationControl_U1Em5".manualOperationEmArea,
                           manualOperationCms := "ManualOperationControl_U1Em5".manualOperationCms,
                           Axis := "ManualOperationControl_U1Em5".axis,
                           Axis64Pos := "ManualOperationControl_U1Em5".axis64Pos,
                           AxisSfotCam := "ManualOperationControl_U1Em5".softCam,
                           Sina := "ManualOperationControl_U1Em5".sina,
                           twoWayAcutor := "ManualOperationControl_U1Em5".twoWayActuator,
                           Status := #StatusEm[5].Status,
                           errorID := #errorIDEm[5].errorID);
END_REGION

REGION Network 14 (SCL): Equipment Module 6 Cms Mapping
   REGION Input Mapping
       // Axis
       "ManualOperationControl_U1Em6".axis64Pos[1].monitoring := "Unit1.Em6.HmiInterface".cmVisionUnitAxisZ.monitoring;

       // SoftCam
       "ManualOperationControl_U1Em6".softCam[1] := "Unit1.Em6.HmiInterface".cm.softcam.visionUnit;

       // TwoWayActuator
       "ManualOperationControl_U1Em6".twoWayActuator[1].monitoring := "Unit1.Em6.HmiInterface".cmVisionPusherSupportUpDown.monitoring;
   END_REGION


   REGION Output Mapping
       // Axis
       "CallManualOperationLines_ServoPos64Commands"(ManualOperationControl := "ManualOperationControl_U1Em6".axis64Pos[1].commands,
                                                     HmiInterface => "Unit1.Em6.HmiInterface".cmVisionUnitAxisZ.commands);

       // TwoWayActuator
       "Unit1.Em6.HmiInterface".cmVisionPusherSupportUpDown.commands := "ManualOperationControl_U1Em6".twoWayActuator[1].commands;
   END_REGION
END_REGION

REGION Network 15: Equipment Module 6
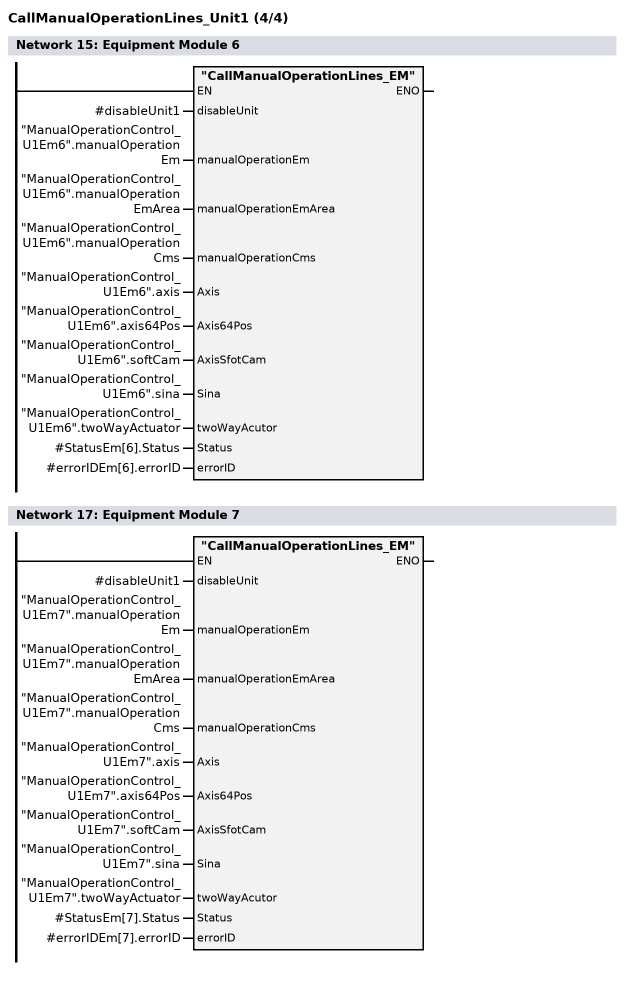
   RUNG wire#powerrail
      "CallManualOperationLines_EM"(disableUnit := #disableUnit1, manualOperationEm := "ManualOperationControl_U1Em6".manualOperationEm, manualOperationEmArea := "ManualOperationControl_U1Em6".manualOperationEmArea, manualOperationCms := "ManualOperationControl_U1Em6".manualOperationCms, Axis := "ManualOperationControl_U1Em6".axis, Axis64Pos := "ManualOperationControl_U1Em6".axis64Pos, AxisSfotCam := "ManualOperationControl_U1Em6".softCam, Sina := "ManualOperationControl_U1Em6".sina, twoWayAcutor := "ManualOperationControl_U1Em6".twoWayActuator, Status := #StatusEm[6].Status, errorID := #errorIDEm[6].errorID)
   END_RUNG
   // the same network as SCL:
   "CallManualOperationLines_EM"(disableUnit := #disableUnit1,
                           manualOperationEm := "ManualOperationControl_U1Em6".manualOperationEm,
                           manualOperationEmArea := "ManualOperationControl_U1Em6".manualOperationEmArea,
                           manualOperationCms := "ManualOperationControl_U1Em6".manualOperationCms,
                           Axis := "ManualOperationControl_U1Em6".axis,
                           Axis64Pos := "ManualOperationControl_U1Em6".axis64Pos,
                           AxisSfotCam := "ManualOperationControl_U1Em6".softCam,
                           Sina := "ManualOperationControl_U1Em6".sina,
                           twoWayAcutor := "ManualOperationControl_U1Em6".twoWayActuator,
                           Status := #StatusEm[6].Status,
                           errorID := #errorIDEm[6].errorID);
END_REGION

REGION Network 16 (SCL): Equipment Module 7 Cms Mapping
   REGION Input Mapping
       // Axis
       "ManualOperationControl_U1Em7".axis[1].monitoring := "Unit1.Em7.HmiInterface".cmNgKickerAxisZ.monitoring;
       "ManualOperationControl_U1Em7".axis[2].monitoring := "Unit1.Em7.HmiInterface".cmPassKickerAxisZ.monitoring;
       "ManualOperationControl_U1Em7".axis[3].monitoring := "Unit1.Em7.HmiInterface".cmCutConveyorAxisB.monitoring;
       "ManualOperationControl_U1Em7".axis[4].monitoring := "Unit1.Em7.HmiInterface".cmNgConveyorAxisB.monitoring;
       "ManualOperationControl_U1Em7".axis[5].monitoring := "Unit1.Em7.HmiInterface".cmStack1ConveyorAxisB.monitoring;
       "ManualOperationControl_U1Em7".axis[6].monitoring := "Unit1.Em7.HmiInterface".cmStack2ConveyorAxisB.monitoring;

       // Sina Speed
       "ManualOperationControl_U1Em7".sina[1].monitoring := "Unit1.Em7.HmiInterface".cmCutConveyorRingBlow.monitoring;
       "ManualOperationControl_U1Em7".sina[2].monitoring := "Unit1.Em7.HmiInterface".cmNgConveyorRingBlow.monitoring;
       "ManualOperationControl_U1Em7".sina[3].monitoring := "Unit1.Em7.HmiInterface".cmStack2ConveyorRingBlow.monitoring;

       // TwoWayActuator
       "ManualOperationControl_U1Em7".twoWayActuator[1].monitoring := "Unit1.Em7.HmiInterface".cmNgBoxLockCylinderUpDown.monitoring;
   END_REGION


   REGION Output Mapping
       // Axis
       "CallManualOperationLines_ServoCommands"(ManualOperationControl := "ManualOperationControl_U1Em7".axis[1].commands,
                                                HmiInterface => "Unit1.Em7.HmiInterface".cmNgKickerAxisZ.commands);
       "CallManualOperationLines_ServoCommands"(ManualOperationControl := "ManualOperationControl_U1Em7".axis[2].commands,
                                                HmiInterface => "Unit1.Em7.HmiInterface".cmPassKickerAxisZ.commands);
       "CallManualOperationLines_ServoCommands"(ManualOperationControl := "ManualOperationControl_U1Em7".axis[3].commands,
                                                HmiInterface => "Unit1.Em7.HmiInterface".cmCutConveyorAxisB.commands);
       "CallManualOperationLines_ServoCommands"(ManualOperationControl := "ManualOperationControl_U1Em7".axis[4].commands,
                                                HmiInterface => "Unit1.Em7.HmiInterface".cmNgConveyorAxisB.commands);
       "CallManualOperationLines_ServoCommands"(ManualOperationControl := "ManualOperationControl_U1Em7".axis[5].commands,
                                                HmiInterface => "Unit1.Em7.HmiInterface".cmStack1ConveyorAxisB.commands);
       "CallManualOperationLines_ServoCommands"(ManualOperationControl := "ManualOperationControl_U1Em7".axis[6].commands,
                                                HmiInterface => "Unit1.Em7.HmiInterface".cmStack2ConveyorAxisB.commands);

       // Sina Speed
       "Unit1.Em7.HmiInterface".cmCutConveyorRingBlow.commands.moveVelocity := "ManualOperationControl_U1Em7".sina[1].commands.moveVelocity;
       "Unit1.Em7.HmiInterface".cmCutConveyorRingBlow.commands.stop := "ManualOperationControl_U1Em7".sina[1].commands.stop;
       "Unit1.Em7.HmiInterface".cmNgConveyorRingBlow.commands.moveVelocity := "ManualOperationControl_U1Em7".sina[2].commands.moveVelocity;
       "Unit1.Em7.HmiInterface".cmNgConveyorRingBlow.commands.stop := "ManualOperationControl_U1Em7".sina[2].commands.stop;
       "Unit1.Em7.HmiInterface".cmStack2ConveyorRingBlow.commands.moveVelocity := "ManualOperationControl_U1Em7".sina[3].commands.moveVelocity;
       "Unit1.Em7.HmiInterface".cmStack2ConveyorRingBlow.commands.stop := "ManualOperationControl_U1Em7".sina[3].commands.stop;

       // TwoWayActuator
       "Unit1.Em7.HmiInterface".cmNgBoxLockCylinderUpDown.commands := "ManualOperationControl_U1Em7".twoWayActuator[1].commands;
   END_REGION
END_REGION

REGION Network 17: Equipment Module 7
   RUNG wire#powerrail
      "CallManualOperationLines_EM"(disableUnit := #disableUnit1, manualOperationEm := "ManualOperationControl_U1Em7".manualOperationEm, manualOperationEmArea := "ManualOperationControl_U1Em7".manualOperationEmArea, manualOperationCms := "ManualOperationControl_U1Em7".manualOperationCms, Axis := "ManualOperationControl_U1Em7".axis, Axis64Pos := "ManualOperationControl_U1Em7".axis64Pos, AxisSfotCam := "ManualOperationControl_U1Em7".softCam, Sina := "ManualOperationControl_U1Em7".sina, twoWayAcutor := "ManualOperationControl_U1Em7".twoWayActuator, Status := #StatusEm[7].Status, errorID := #errorIDEm[7].errorID)
   END_RUNG
   // the same network as SCL:
   "CallManualOperationLines_EM"(disableUnit := #disableUnit1,
                           manualOperationEm := "ManualOperationControl_U1Em7".manualOperationEm,
                           manualOperationEmArea := "ManualOperationControl_U1Em7".manualOperationEmArea,
                           manualOperationCms := "ManualOperationControl_U1Em7".manualOperationCms,
                           Axis := "ManualOperationControl_U1Em7".axis,
                           Axis64Pos := "ManualOperationControl_U1Em7".axis64Pos,
                           AxisSfotCam := "ManualOperationControl_U1Em7".softCam,
                           Sina := "ManualOperationControl_U1Em7".sina,
                           twoWayAcutor := "ManualOperationControl_U1Em7".twoWayActuator,
                           Status := #StatusEm[7].Status,
                           errorID := #errorIDEm[7].errorID);
END_REGION
END_FUNCTION

FUNCTION "CallManualOperationLines_EM" : Void   // FC66, LAD
// stored: SetENOAutomatically false
   VAR_INPUT
      disableUnit : Bool;
   END_VAR
   VAR_IN_OUT
      manualOperationEm : "LAF_typeManEm";
      manualOperationEmArea : Array[*] of "LAF_typeManOperationArea";
      manualOperationCms : Array[*] of "LAF_typeManOperation";
      Axis : Array[*] of "LBC_typeAxisControlInterface";
      Axis64Pos : Array[*] of "LBC_typeAxis64PosInterface";
      AxisSfotCam : Array[*] of "LER_typeSoftCamRelation";
      Sina : Array[*] of "LBC_typeSinaSpeedInterface";
      twoWayAcutor : Array[*] of "LBC_typeTwoWayActuatorInterface";
      Status : Array[*] of Word;
      errorID : Array[*] of Word;
   END_VAR
   VAR_TEMP
      tempLowerBoundAxis : Int;
      tempUpperBoundAxis : Int;
      tempLowerBoundAxis64Pos : Int;
      tempUpperBoundAxis64Pos : Int;
      tempLowerBoundSina : Int;
      tempUpperBoundSina : Int;
      tempLowerBoundTwoWayAct : Int;
      tempUpperBoundTwoWayAct : Int;
      tempEnd : Bool;
   END_VAR
BEGIN

REGION Network 1: Detect lower and upper bound of the array for further processing
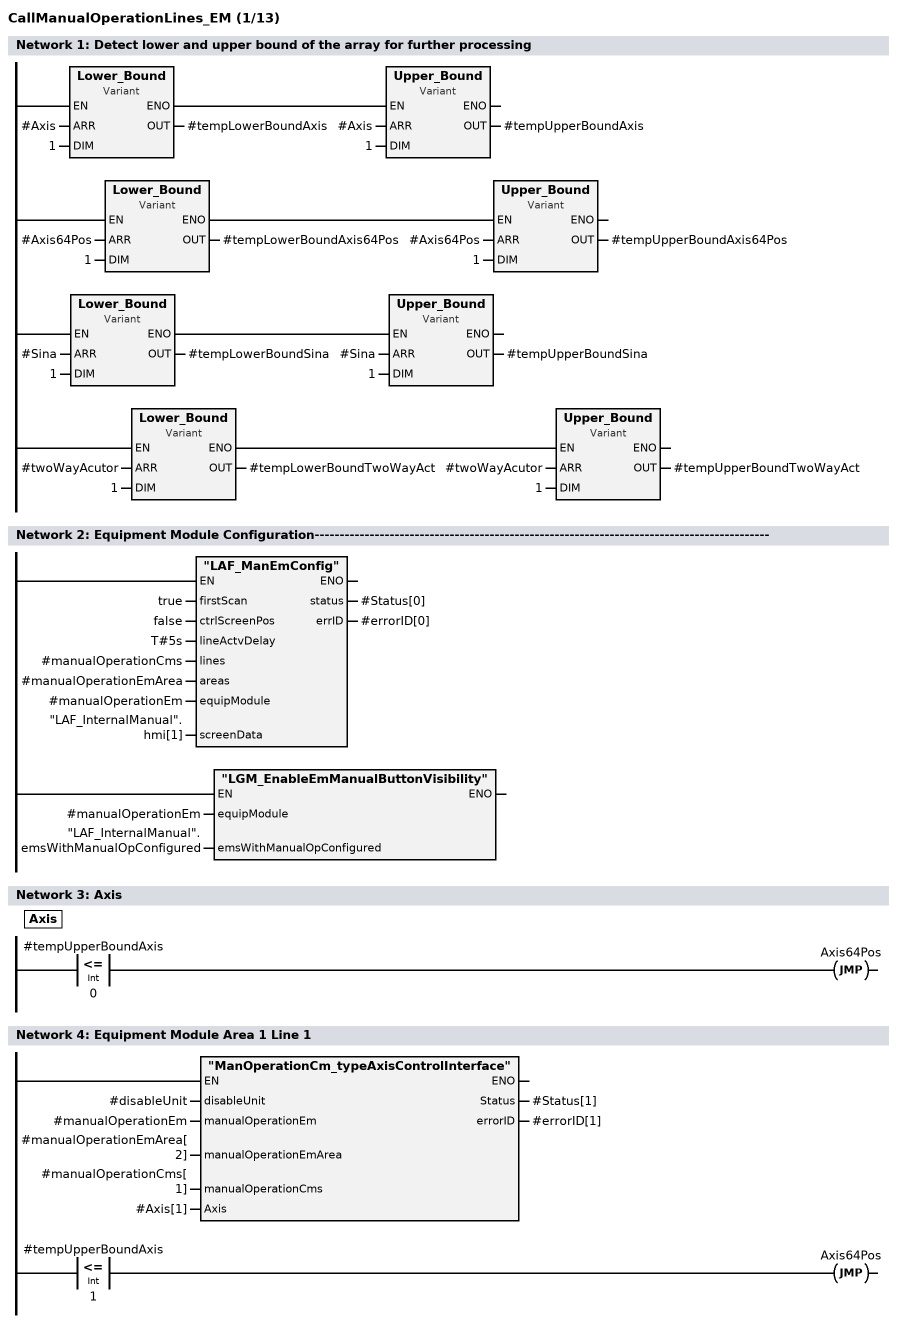
   // no SCL statement known for Lower_Bound, Upper_Bound: written as a call
   // ENO of a box is taken as its EN; it also drops when the box reports an error
   Lower_Bound(arr := #Axis, dim := 1, out => #tempLowerBoundAxis);
   Upper_Bound(arr := #Axis, dim := 1, out => #tempUpperBoundAxis);
   Lower_Bound(arr := #Axis64Pos, dim := 1, out => #tempLowerBoundAxis64Pos);
   Upper_Bound(arr := #Axis64Pos, dim := 1, out => #tempUpperBoundAxis64Pos);
   Lower_Bound(arr := #Sina, dim := 1, out => #tempLowerBoundSina);
   Upper_Bound(arr := #Sina, dim := 1, out => #tempUpperBoundSina);
   Lower_Bound(arr := #twoWayAcutor, dim := 1, out => #tempLowerBoundTwoWayAct);
   Upper_Bound(arr := #twoWayAcutor, dim := 1, out => #tempUpperBoundTwoWayAct);
END_REGION

REGION Network 2: Equipment Module Configuration-------------------------------------------------------------------------------------------
   RUNG wire#powerrail
      "LAF_ManEmConfig"(firstScan := true, ctrlScreenPos := false, lineActvDelay := T#5s, lines := #manualOperationCms, areas := #manualOperationEmArea, equipModule := #manualOperationEm, screenData := "LAF_InternalManual".hmi[1], status => #Status[0], errID => #errorID[0])
   END_RUNG
   RUNG wire#powerrail
      "LGM_EnableEmManualButtonVisibility"(equipModule := #manualOperationEm, emsWithManualOpConfigured := "LAF_InternalManual".emsWithManualOpConfigured)
   END_RUNG
   // the same network as SCL:
   "LAF_ManEmConfig"(firstScan := true,
                     ctrlScreenPos := false,
                     lineActvDelay := T#5s,
                     lines := #manualOperationCms,
                     areas := #manualOperationEmArea,
                     equipModule := #manualOperationEm,
                     screenData := "LAF_InternalManual".hmi[1],
                     status => #Status[0],
                     errID => #errorID[0]);
   "LGM_EnableEmManualButtonVisibility"(equipModule := #manualOperationEm,
                           emsWithManualOpConfigured := "LAF_InternalManual".emsWithManualOpConfigured);
END_REGION

REGION Network 3: Axis
   Label( Axis )
   RUNG wire#powerrail
      { S7_Templates := "SrcType := Int" } LE_Contact(in1 := #tempUpperBoundAxis, in2 := 0)
      JumpCoil( Axis64Pos )
   END_RUNG
   // the same network as SCL:
   Axis:
   IF #tempUpperBoundAxis <= 0 THEN GOTO Axis64Pos; END_IF;
END_REGION

REGION Network 4: Equipment Module Area 1 Line 1
   RUNG wire#powerrail
      "ManOperationCm_typeAxisControlInterface"(disableUnit := #disableUnit, manualOperationEm := #manualOperationEm, manualOperationEmArea := #manualOperationEmArea[2], manualOperationCms := #manualOperationCms[1], Axis := #Axis[1], Status => #Status[1], errorID => #errorID[1])
   END_RUNG
   RUNG wire#powerrail
      { S7_Templates := "SrcType := Int" } LE_Contact(in1 := #tempUpperBoundAxis, in2 := 1)
      JumpCoil( Axis64Pos )
   END_RUNG
   // the same network as SCL:
   "ManOperationCm_typeAxisControlInterface"(disableUnit := #disableUnit,
                           manualOperationEm := #manualOperationEm,
                           manualOperationEmArea := #manualOperationEmArea[2],
                           manualOperationCms := #manualOperationCms[1],
                           Axis := #Axis[1],
                           Status => #Status[1],
                           errorID => #errorID[1]);
   IF #tempUpperBoundAxis <= 1 THEN GOTO Axis64Pos; END_IF;
END_REGION

REGION Network 5: Equipment Module Area 1 Line 2
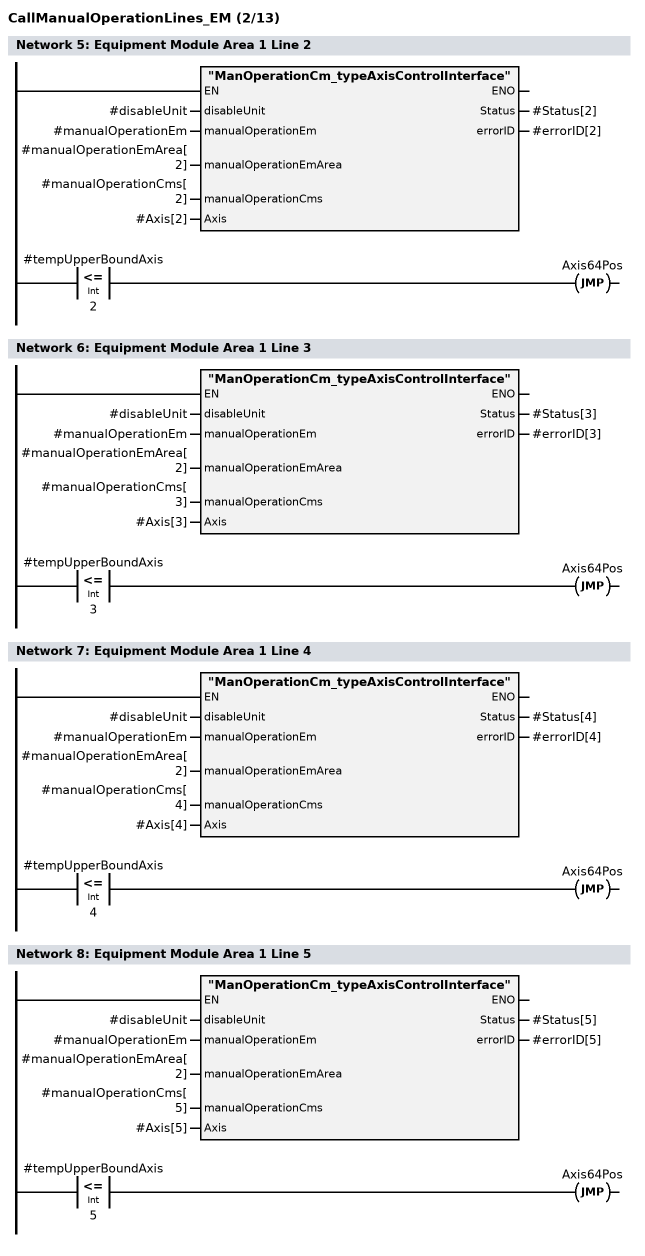
   RUNG wire#powerrail
      "ManOperationCm_typeAxisControlInterface"(disableUnit := #disableUnit, manualOperationEm := #manualOperationEm, manualOperationEmArea := #manualOperationEmArea[2], manualOperationCms := #manualOperationCms[2], Axis := #Axis[2], Status => #Status[2], errorID => #errorID[2])
   END_RUNG
   RUNG wire#powerrail
      { S7_Templates := "SrcType := Int" } LE_Contact(in1 := #tempUpperBoundAxis, in2 := 2)
      JumpCoil( Axis64Pos )
   END_RUNG
   // the same network as SCL:
   "ManOperationCm_typeAxisControlInterface"(disableUnit := #disableUnit,
                           manualOperationEm := #manualOperationEm,
                           manualOperationEmArea := #manualOperationEmArea[2],
                           manualOperationCms := #manualOperationCms[2],
                           Axis := #Axis[2],
                           Status => #Status[2],
                           errorID => #errorID[2]);
   IF #tempUpperBoundAxis <= 2 THEN GOTO Axis64Pos; END_IF;
END_REGION

REGION Network 6: Equipment Module Area 1 Line 3
   RUNG wire#powerrail
      "ManOperationCm_typeAxisControlInterface"(disableUnit := #disableUnit, manualOperationEm := #manualOperationEm, manualOperationEmArea := #manualOperationEmArea[2], manualOperationCms := #manualOperationCms[3], Axis := #Axis[3], Status => #Status[3], errorID => #errorID[3])
   END_RUNG
   RUNG wire#powerrail
      { S7_Templates := "SrcType := Int" } LE_Contact(in1 := #tempUpperBoundAxis, in2 := 3)
      JumpCoil( Axis64Pos )
   END_RUNG
   // the same network as SCL:
   "ManOperationCm_typeAxisControlInterface"(disableUnit := #disableUnit,
                           manualOperationEm := #manualOperationEm,
                           manualOperationEmArea := #manualOperationEmArea[2],
                           manualOperationCms := #manualOperationCms[3],
                           Axis := #Axis[3],
                           Status => #Status[3],
                           errorID => #errorID[3]);
   IF #tempUpperBoundAxis <= 3 THEN GOTO Axis64Pos; END_IF;
END_REGION

REGION Network 7: Equipment Module Area 1 Line 4
   RUNG wire#powerrail
      "ManOperationCm_typeAxisControlInterface"(disableUnit := #disableUnit, manualOperationEm := #manualOperationEm, manualOperationEmArea := #manualOperationEmArea[2], manualOperationCms := #manualOperationCms[4], Axis := #Axis[4], Status => #Status[4], errorID => #errorID[4])
   END_RUNG
   RUNG wire#powerrail
      { S7_Templates := "SrcType := Int" } LE_Contact(in1 := #tempUpperBoundAxis, in2 := 4)
      JumpCoil( Axis64Pos )
   END_RUNG
   // the same network as SCL:
   "ManOperationCm_typeAxisControlInterface"(disableUnit := #disableUnit,
                           manualOperationEm := #manualOperationEm,
                           manualOperationEmArea := #manualOperationEmArea[2],
                           manualOperationCms := #manualOperationCms[4],
                           Axis := #Axis[4],
                           Status => #Status[4],
                           errorID => #errorID[4]);
   IF #tempUpperBoundAxis <= 4 THEN GOTO Axis64Pos; END_IF;
END_REGION

REGION Network 8: Equipment Module Area 1 Line 5
   RUNG wire#powerrail
      "ManOperationCm_typeAxisControlInterface"(disableUnit := #disableUnit, manualOperationEm := #manualOperationEm, manualOperationEmArea := #manualOperationEmArea[2], manualOperationCms := #manualOperationCms[5], Axis := #Axis[5], Status => #Status[5], errorID => #errorID[5])
   END_RUNG
   RUNG wire#powerrail
      { S7_Templates := "SrcType := Int" } LE_Contact(in1 := #tempUpperBoundAxis, in2 := 5)
      JumpCoil( Axis64Pos )
   END_RUNG
   // the same network as SCL:
   "ManOperationCm_typeAxisControlInterface"(disableUnit := #disableUnit,
                           manualOperationEm := #manualOperationEm,
                           manualOperationEmArea := #manualOperationEmArea[2],
                           manualOperationCms := #manualOperationCms[5],
                           Axis := #Axis[5],
                           Status => #Status[5],
                           errorID => #errorID[5]);
   IF #tempUpperBoundAxis <= 5 THEN GOTO Axis64Pos; END_IF;
END_REGION

REGION Network 9: Equipment Module Area 1 Line 6
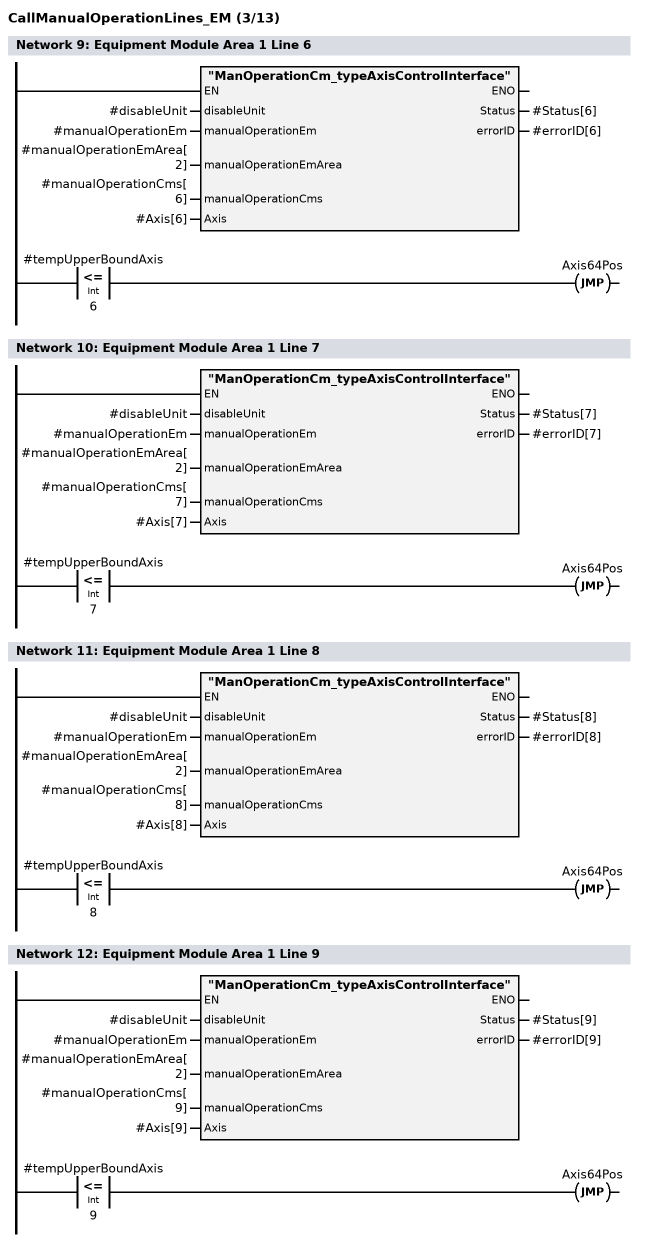
   RUNG wire#powerrail
      "ManOperationCm_typeAxisControlInterface"(disableUnit := #disableUnit, manualOperationEm := #manualOperationEm, manualOperationEmArea := #manualOperationEmArea[2], manualOperationCms := #manualOperationCms[6], Axis := #Axis[6], Status => #Status[6], errorID => #errorID[6])
   END_RUNG
   RUNG wire#powerrail
      { S7_Templates := "SrcType := Int" } LE_Contact(in1 := #tempUpperBoundAxis, in2 := 6)
      JumpCoil( Axis64Pos )
   END_RUNG
   // the same network as SCL:
   "ManOperationCm_typeAxisControlInterface"(disableUnit := #disableUnit,
                           manualOperationEm := #manualOperationEm,
                           manualOperationEmArea := #manualOperationEmArea[2],
                           manualOperationCms := #manualOperationCms[6],
                           Axis := #Axis[6],
                           Status => #Status[6],
                           errorID => #errorID[6]);
   IF #tempUpperBoundAxis <= 6 THEN GOTO Axis64Pos; END_IF;
END_REGION

REGION Network 10: Equipment Module Area 1 Line 7
   RUNG wire#powerrail
      "ManOperationCm_typeAxisControlInterface"(disableUnit := #disableUnit, manualOperationEm := #manualOperationEm, manualOperationEmArea := #manualOperationEmArea[2], manualOperationCms := #manualOperationCms[7], Axis := #Axis[7], Status => #Status[7], errorID => #errorID[7])
   END_RUNG
   RUNG wire#powerrail
      { S7_Templates := "SrcType := Int" } LE_Contact(in1 := #tempUpperBoundAxis, in2 := 7)
      JumpCoil( Axis64Pos )
   END_RUNG
   // the same network as SCL:
   "ManOperationCm_typeAxisControlInterface"(disableUnit := #disableUnit,
                           manualOperationEm := #manualOperationEm,
                           manualOperationEmArea := #manualOperationEmArea[2],
                           manualOperationCms := #manualOperationCms[7],
                           Axis := #Axis[7],
                           Status => #Status[7],
                           errorID => #errorID[7]);
   IF #tempUpperBoundAxis <= 7 THEN GOTO Axis64Pos; END_IF;
END_REGION

REGION Network 11: Equipment Module Area 1 Line 8
   RUNG wire#powerrail
      "ManOperationCm_typeAxisControlInterface"(disableUnit := #disableUnit, manualOperationEm := #manualOperationEm, manualOperationEmArea := #manualOperationEmArea[2], manualOperationCms := #manualOperationCms[8], Axis := #Axis[8], Status => #Status[8], errorID => #errorID[8])
   END_RUNG
   RUNG wire#powerrail
      { S7_Templates := "SrcType := Int" } LE_Contact(in1 := #tempUpperBoundAxis, in2 := 8)
      JumpCoil( Axis64Pos )
   END_RUNG
   // the same network as SCL:
   "ManOperationCm_typeAxisControlInterface"(disableUnit := #disableUnit,
                           manualOperationEm := #manualOperationEm,
                           manualOperationEmArea := #manualOperationEmArea[2],
                           manualOperationCms := #manualOperationCms[8],
                           Axis := #Axis[8],
                           Status => #Status[8],
                           errorID => #errorID[8]);
   IF #tempUpperBoundAxis <= 8 THEN GOTO Axis64Pos; END_IF;
END_REGION

REGION Network 12: Equipment Module Area 1 Line 9
   RUNG wire#powerrail
      "ManOperationCm_typeAxisControlInterface"(disableUnit := #disableUnit, manualOperationEm := #manualOperationEm, manualOperationEmArea := #manualOperationEmArea[2], manualOperationCms := #manualOperationCms[9], Axis := #Axis[9], Status => #Status[9], errorID => #errorID[9])
   END_RUNG
   RUNG wire#powerrail
      { S7_Templates := "SrcType := Int" } LE_Contact(in1 := #tempUpperBoundAxis, in2 := 9)
      JumpCoil( Axis64Pos )
   END_RUNG
   // the same network as SCL:
   "ManOperationCm_typeAxisControlInterface"(disableUnit := #disableUnit,
                           manualOperationEm := #manualOperationEm,
                           manualOperationEmArea := #manualOperationEmArea[2],
                           manualOperationCms := #manualOperationCms[9],
                           Axis := #Axis[9],
                           Status => #Status[9],
                           errorID => #errorID[9]);
   IF #tempUpperBoundAxis <= 9 THEN GOTO Axis64Pos; END_IF;
END_REGION

REGION Network 13: Equipment Module Area 1 Line 10
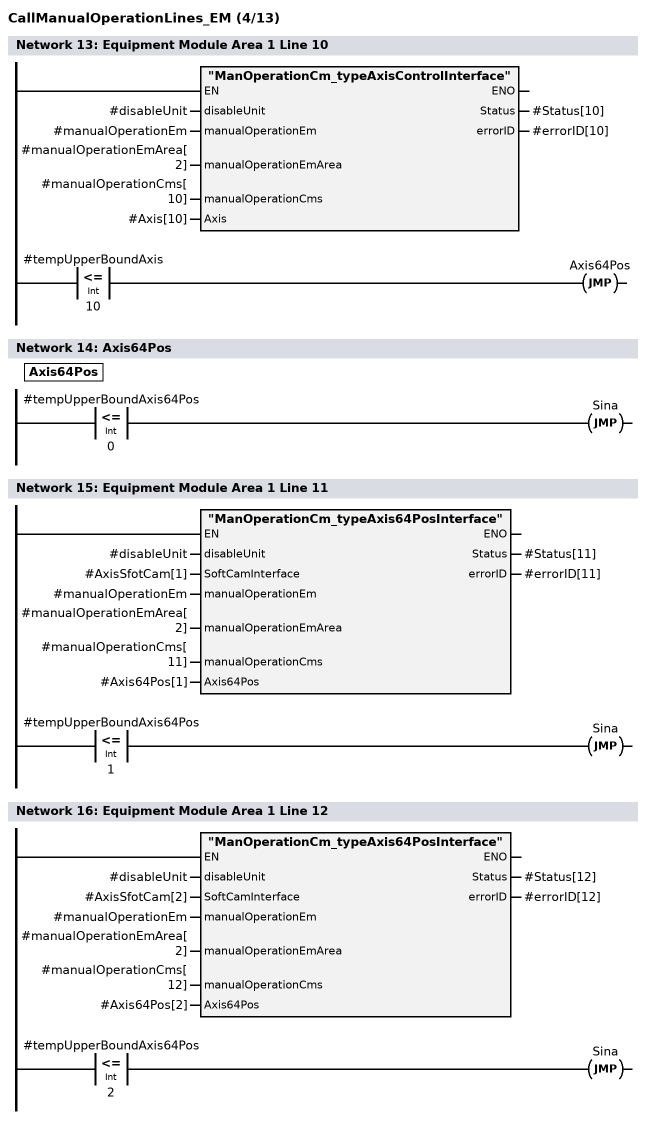
   RUNG wire#powerrail
      "ManOperationCm_typeAxisControlInterface"(disableUnit := #disableUnit, manualOperationEm := #manualOperationEm, manualOperationEmArea := #manualOperationEmArea[2], manualOperationCms := #manualOperationCms[10], Axis := #Axis[10], Status => #Status[10], errorID => #errorID[10])
   END_RUNG
   RUNG wire#powerrail
      { S7_Templates := "SrcType := Int" } LE_Contact(in1 := #tempUpperBoundAxis, in2 := 10)
      JumpCoil( Axis64Pos )
   END_RUNG
   // the same network as SCL:
   "ManOperationCm_typeAxisControlInterface"(disableUnit := #disableUnit,
                           manualOperationEm := #manualOperationEm,
                           manualOperationEmArea := #manualOperationEmArea[2],
                           manualOperationCms := #manualOperationCms[10],
                           Axis := #Axis[10],
                           Status => #Status[10],
                           errorID => #errorID[10]);
   IF #tempUpperBoundAxis <= 10 THEN GOTO Axis64Pos; END_IF;
END_REGION

REGION Network 14: Axis64Pos
   Label( Axis64Pos )
   RUNG wire#powerrail
      { S7_Templates := "SrcType := Int" } LE_Contact(in1 := #tempUpperBoundAxis64Pos, in2 := 0)
      JumpCoil( Sina )
   END_RUNG
   // the same network as SCL:
   Axis64Pos:
   IF #tempUpperBoundAxis64Pos <= 0 THEN GOTO Sina; END_IF;
END_REGION

REGION Network 15: Equipment Module Area 1 Line 11
   RUNG wire#powerrail
      "ManOperationCm_typeAxis64PosInterface"(disableUnit := #disableUnit, SoftCamInterface := #AxisSfotCam[1], manualOperationEm := #manualOperationEm, manualOperationEmArea := #manualOperationEmArea[2], manualOperationCms := #manualOperationCms[11], Axis64Pos := #Axis64Pos[1], Status => #Status[11], errorID => #errorID[11])
   END_RUNG
   RUNG wire#powerrail
      { S7_Templates := "SrcType := Int" } LE_Contact(in1 := #tempUpperBoundAxis64Pos, in2 := 1)
      JumpCoil( Sina )
   END_RUNG
   // the same network as SCL:
   "ManOperationCm_typeAxis64PosInterface"(disableUnit := #disableUnit,
                           SoftCamInterface := #AxisSfotCam[1],
                           manualOperationEm := #manualOperationEm,
                           manualOperationEmArea := #manualOperationEmArea[2],
                           manualOperationCms := #manualOperationCms[11],
                           Axis64Pos := #Axis64Pos[1],
                           Status => #Status[11],
                           errorID => #errorID[11]);
   IF #tempUpperBoundAxis64Pos <= 1 THEN GOTO Sina; END_IF;
END_REGION

REGION Network 16: Equipment Module Area 1 Line 12
   RUNG wire#powerrail
      "ManOperationCm_typeAxis64PosInterface"(disableUnit := #disableUnit, SoftCamInterface := #AxisSfotCam[2], manualOperationEm := #manualOperationEm, manualOperationEmArea := #manualOperationEmArea[2], manualOperationCms := #manualOperationCms[12], Axis64Pos := #Axis64Pos[2], Status => #Status[12], errorID => #errorID[12])
   END_RUNG
   RUNG wire#powerrail
      { S7_Templates := "SrcType := Int" } LE_Contact(in1 := #tempUpperBoundAxis64Pos, in2 := 2)
      JumpCoil( Sina )
   END_RUNG
   // the same network as SCL:
   "ManOperationCm_typeAxis64PosInterface"(disableUnit := #disableUnit,
                           SoftCamInterface := #AxisSfotCam[2],
                           manualOperationEm := #manualOperationEm,
                           manualOperationEmArea := #manualOperationEmArea[2],
                           manualOperationCms := #manualOperationCms[12],
                           Axis64Pos := #Axis64Pos[2],
                           Status => #Status[12],
                           errorID => #errorID[12]);
   IF #tempUpperBoundAxis64Pos <= 2 THEN GOTO Sina; END_IF;
END_REGION

REGION Network 17: Equipment Module Area 1 Line 13
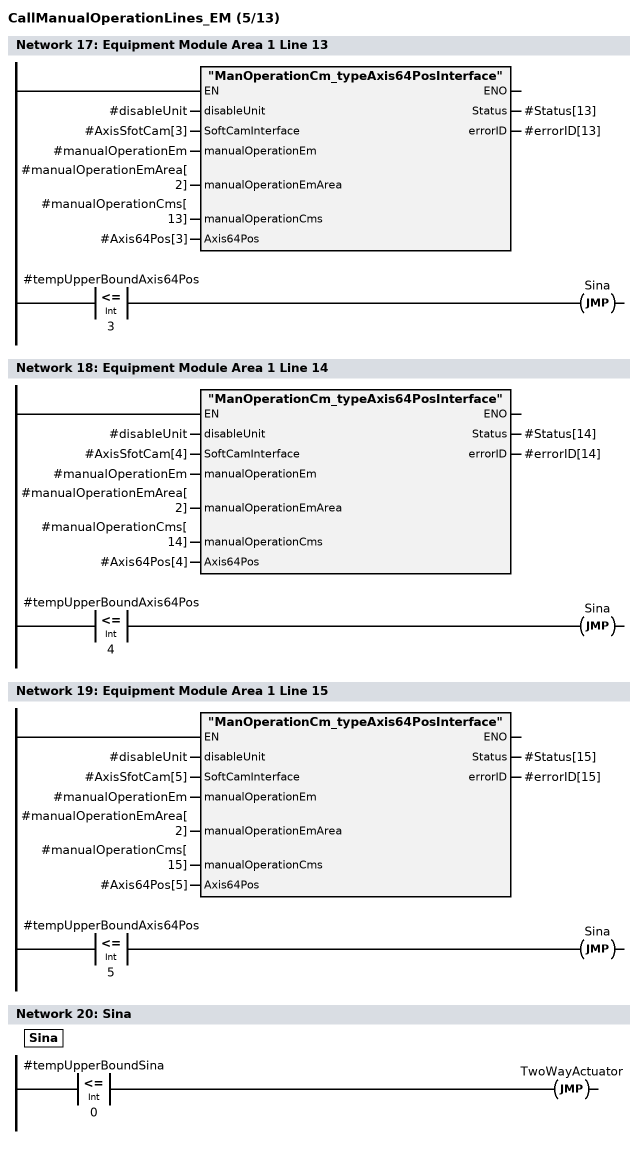
   RUNG wire#powerrail
      "ManOperationCm_typeAxis64PosInterface"(disableUnit := #disableUnit, SoftCamInterface := #AxisSfotCam[3], manualOperationEm := #manualOperationEm, manualOperationEmArea := #manualOperationEmArea[2], manualOperationCms := #manualOperationCms[13], Axis64Pos := #Axis64Pos[3], Status => #Status[13], errorID => #errorID[13])
   END_RUNG
   RUNG wire#powerrail
      { S7_Templates := "SrcType := Int" } LE_Contact(in1 := #tempUpperBoundAxis64Pos, in2 := 3)
      JumpCoil( Sina )
   END_RUNG
   // the same network as SCL:
   "ManOperationCm_typeAxis64PosInterface"(disableUnit := #disableUnit,
                           SoftCamInterface := #AxisSfotCam[3],
                           manualOperationEm := #manualOperationEm,
                           manualOperationEmArea := #manualOperationEmArea[2],
                           manualOperationCms := #manualOperationCms[13],
                           Axis64Pos := #Axis64Pos[3],
                           Status => #Status[13],
                           errorID => #errorID[13]);
   IF #tempUpperBoundAxis64Pos <= 3 THEN GOTO Sina; END_IF;
END_REGION

REGION Network 18: Equipment Module Area 1 Line 14
   RUNG wire#powerrail
      "ManOperationCm_typeAxis64PosInterface"(disableUnit := #disableUnit, SoftCamInterface := #AxisSfotCam[4], manualOperationEm := #manualOperationEm, manualOperationEmArea := #manualOperationEmArea[2], manualOperationCms := #manualOperationCms[14], Axis64Pos := #Axis64Pos[4], Status => #Status[14], errorID => #errorID[14])
   END_RUNG
   RUNG wire#powerrail
      { S7_Templates := "SrcType := Int" } LE_Contact(in1 := #tempUpperBoundAxis64Pos, in2 := 4)
      JumpCoil( Sina )
   END_RUNG
   // the same network as SCL:
   "ManOperationCm_typeAxis64PosInterface"(disableUnit := #disableUnit,
                           SoftCamInterface := #AxisSfotCam[4],
                           manualOperationEm := #manualOperationEm,
                           manualOperationEmArea := #manualOperationEmArea[2],
                           manualOperationCms := #manualOperationCms[14],
                           Axis64Pos := #Axis64Pos[4],
                           Status => #Status[14],
                           errorID => #errorID[14]);
   IF #tempUpperBoundAxis64Pos <= 4 THEN GOTO Sina; END_IF;
END_REGION

REGION Network 19: Equipment Module Area 1 Line 15
   RUNG wire#powerrail
      "ManOperationCm_typeAxis64PosInterface"(disableUnit := #disableUnit, SoftCamInterface := #AxisSfotCam[5], manualOperationEm := #manualOperationEm, manualOperationEmArea := #manualOperationEmArea[2], manualOperationCms := #manualOperationCms[15], Axis64Pos := #Axis64Pos[5], Status => #Status[15], errorID => #errorID[15])
   END_RUNG
   RUNG wire#powerrail
      { S7_Templates := "SrcType := Int" } LE_Contact(in1 := #tempUpperBoundAxis64Pos, in2 := 5)
      JumpCoil( Sina )
   END_RUNG
   // the same network as SCL:
   "ManOperationCm_typeAxis64PosInterface"(disableUnit := #disableUnit,
                           SoftCamInterface := #AxisSfotCam[5],
                           manualOperationEm := #manualOperationEm,
                           manualOperationEmArea := #manualOperationEmArea[2],
                           manualOperationCms := #manualOperationCms[15],
                           Axis64Pos := #Axis64Pos[5],
                           Status => #Status[15],
                           errorID => #errorID[15]);
   IF #tempUpperBoundAxis64Pos <= 5 THEN GOTO Sina; END_IF;
END_REGION

REGION Network 20: Sina
   Label( Sina )
   RUNG wire#powerrail
      { S7_Templates := "SrcType := Int" } LE_Contact(in1 := #tempUpperBoundSina, in2 := 0)
      JumpCoil( TwoWayActuator )
   END_RUNG
   // the same network as SCL:
   Sina:
   IF #tempUpperBoundSina <= 0 THEN GOTO TwoWayActuator; END_IF;
END_REGION

REGION Network 21: Equipment Module Area 1 Line 16
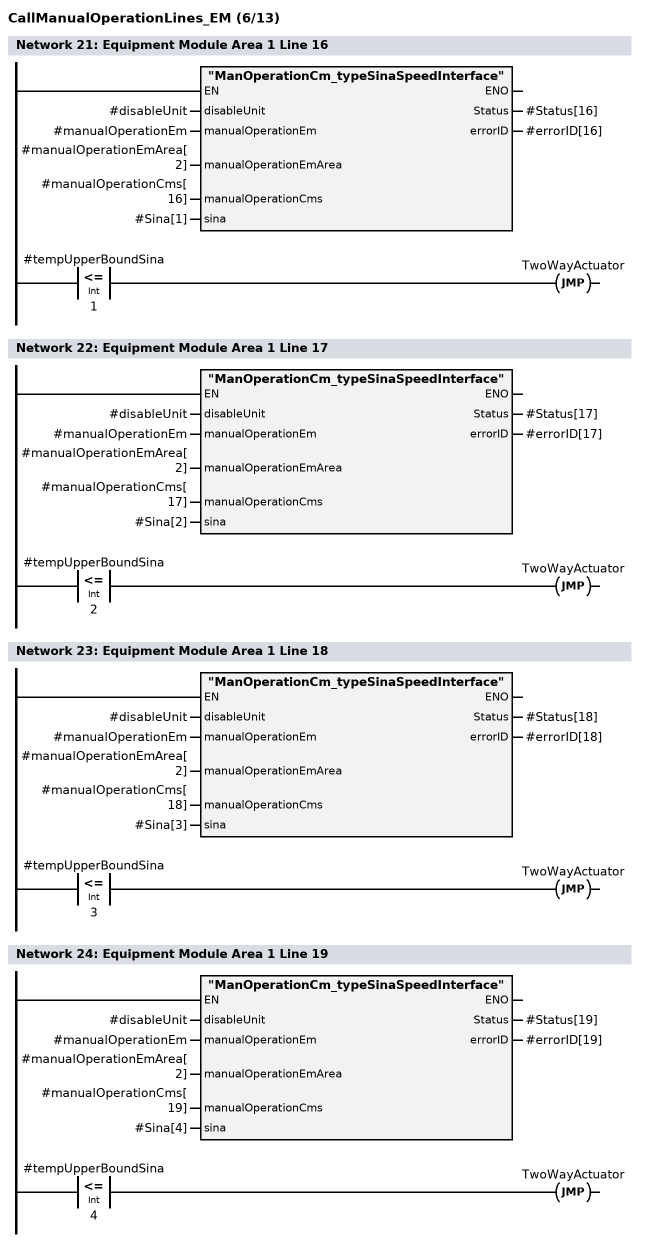
   RUNG wire#powerrail
      "ManOperationCm_typeSinaSpeedInterface"(disableUnit := #disableUnit, manualOperationEm := #manualOperationEm, manualOperationEmArea := #manualOperationEmArea[2], manualOperationCms := #manualOperationCms[16], sina := #Sina[1], Status => #Status[16], errorID => #errorID[16])
   END_RUNG
   RUNG wire#powerrail
      { S7_Templates := "SrcType := Int" } LE_Contact(in1 := #tempUpperBoundSina, in2 := 1)
      JumpCoil( TwoWayActuator )
   END_RUNG
   // the same network as SCL:
   "ManOperationCm_typeSinaSpeedInterface"(disableUnit := #disableUnit,
                           manualOperationEm := #manualOperationEm,
                           manualOperationEmArea := #manualOperationEmArea[2],
                           manualOperationCms := #manualOperationCms[16],
                           sina := #Sina[1],
                           Status => #Status[16],
                           errorID => #errorID[16]);
   IF #tempUpperBoundSina <= 1 THEN GOTO TwoWayActuator; END_IF;
END_REGION

REGION Network 22: Equipment Module Area 1 Line 17
   RUNG wire#powerrail
      "ManOperationCm_typeSinaSpeedInterface"(disableUnit := #disableUnit, manualOperationEm := #manualOperationEm, manualOperationEmArea := #manualOperationEmArea[2], manualOperationCms := #manualOperationCms[17], sina := #Sina[2], Status => #Status[17], errorID => #errorID[17])
   END_RUNG
   RUNG wire#powerrail
      { S7_Templates := "SrcType := Int" } LE_Contact(in1 := #tempUpperBoundSina, in2 := 2)
      JumpCoil( TwoWayActuator )
   END_RUNG
   // the same network as SCL:
   "ManOperationCm_typeSinaSpeedInterface"(disableUnit := #disableUnit,
                           manualOperationEm := #manualOperationEm,
                           manualOperationEmArea := #manualOperationEmArea[2],
                           manualOperationCms := #manualOperationCms[17],
                           sina := #Sina[2],
                           Status => #Status[17],
                           errorID => #errorID[17]);
   IF #tempUpperBoundSina <= 2 THEN GOTO TwoWayActuator; END_IF;
END_REGION

REGION Network 23: Equipment Module Area 1 Line 18
   RUNG wire#powerrail
      "ManOperationCm_typeSinaSpeedInterface"(disableUnit := #disableUnit, manualOperationEm := #manualOperationEm, manualOperationEmArea := #manualOperationEmArea[2], manualOperationCms := #manualOperationCms[18], sina := #Sina[3], Status => #Status[18], errorID => #errorID[18])
   END_RUNG
   RUNG wire#powerrail
      { S7_Templates := "SrcType := Int" } LE_Contact(in1 := #tempUpperBoundSina, in2 := 3)
      JumpCoil( TwoWayActuator )
   END_RUNG
   // the same network as SCL:
   "ManOperationCm_typeSinaSpeedInterface"(disableUnit := #disableUnit,
                           manualOperationEm := #manualOperationEm,
                           manualOperationEmArea := #manualOperationEmArea[2],
                           manualOperationCms := #manualOperationCms[18],
                           sina := #Sina[3],
                           Status => #Status[18],
                           errorID => #errorID[18]);
   IF #tempUpperBoundSina <= 3 THEN GOTO TwoWayActuator; END_IF;
END_REGION

REGION Network 24: Equipment Module Area 1 Line 19
   RUNG wire#powerrail
      "ManOperationCm_typeSinaSpeedInterface"(disableUnit := #disableUnit, manualOperationEm := #manualOperationEm, manualOperationEmArea := #manualOperationEmArea[2], manualOperationCms := #manualOperationCms[19], sina := #Sina[4], Status => #Status[19], errorID => #errorID[19])
   END_RUNG
   RUNG wire#powerrail
      { S7_Templates := "SrcType := Int" } LE_Contact(in1 := #tempUpperBoundSina, in2 := 4)
      JumpCoil( TwoWayActuator )
   END_RUNG
   // the same network as SCL:
   "ManOperationCm_typeSinaSpeedInterface"(disableUnit := #disableUnit,
                           manualOperationEm := #manualOperationEm,
                           manualOperationEmArea := #manualOperationEmArea[2],
                           manualOperationCms := #manualOperationCms[19],
                           sina := #Sina[4],
                           Status => #Status[19],
                           errorID => #errorID[19]);
   IF #tempUpperBoundSina <= 4 THEN GOTO TwoWayActuator; END_IF;
END_REGION

REGION Network 25: Equipment Module Area 1 Line 20
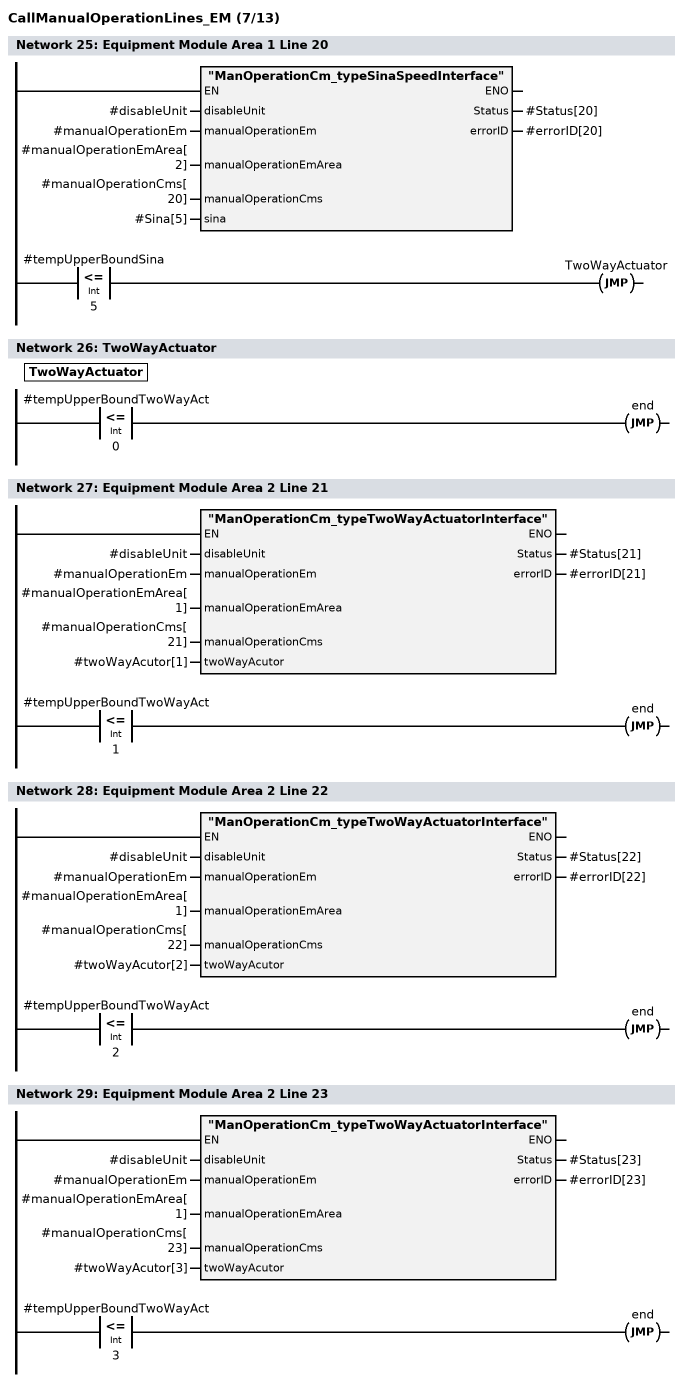
   RUNG wire#powerrail
      "ManOperationCm_typeSinaSpeedInterface"(disableUnit := #disableUnit, manualOperationEm := #manualOperationEm, manualOperationEmArea := #manualOperationEmArea[2], manualOperationCms := #manualOperationCms[20], sina := #Sina[5], Status => #Status[20], errorID => #errorID[20])
   END_RUNG
   RUNG wire#powerrail
      { S7_Templates := "SrcType := Int" } LE_Contact(in1 := #tempUpperBoundSina, in2 := 5)
      JumpCoil( TwoWayActuator )
   END_RUNG
   // the same network as SCL:
   "ManOperationCm_typeSinaSpeedInterface"(disableUnit := #disableUnit,
                           manualOperationEm := #manualOperationEm,
                           manualOperationEmArea := #manualOperationEmArea[2],
                           manualOperationCms := #manualOperationCms[20],
                           sina := #Sina[5],
                           Status => #Status[20],
                           errorID => #errorID[20]);
   IF #tempUpperBoundSina <= 5 THEN GOTO TwoWayActuator; END_IF;
END_REGION

REGION Network 26: TwoWayActuator
   Label( TwoWayActuator )
   RUNG wire#powerrail
      { S7_Templates := "SrcType := Int" } LE_Contact(in1 := #tempUpperBoundTwoWayAct, in2 := 0)
      JumpCoil( end )
   END_RUNG
   // the same network as SCL:
   TwoWayActuator:
   IF #tempUpperBoundTwoWayAct <= 0 THEN GOTO end; END_IF;
END_REGION

REGION Network 27: Equipment Module Area 2 Line 21
   RUNG wire#powerrail
      "ManOperationCm_typeTwoWayActuatorInterface"(disableUnit := #disableUnit, manualOperationEm := #manualOperationEm, manualOperationEmArea := #manualOperationEmArea[1], manualOperationCms := #manualOperationCms[21], twoWayAcutor := #twoWayAcutor[1], Status => #Status[21], errorID => #errorID[21])
   END_RUNG
   RUNG wire#powerrail
      { S7_Templates := "SrcType := Int" } LE_Contact(in1 := #tempUpperBoundTwoWayAct, in2 := 1)
      JumpCoil( end )
   END_RUNG
   // the same network as SCL:
   "ManOperationCm_typeTwoWayActuatorInterface"(disableUnit := #disableUnit,
                           manualOperationEm := #manualOperationEm,
                           manualOperationEmArea := #manualOperationEmArea[1],
                           manualOperationCms := #manualOperationCms[21],
                           twoWayAcutor := #twoWayAcutor[1],
                           Status => #Status[21],
                           errorID => #errorID[21]);
   IF #tempUpperBoundTwoWayAct <= 1 THEN GOTO end; END_IF;
END_REGION

REGION Network 28: Equipment Module Area 2 Line 22
   RUNG wire#powerrail
      "ManOperationCm_typeTwoWayActuatorInterface"(disableUnit := #disableUnit, manualOperationEm := #manualOperationEm, manualOperationEmArea := #manualOperationEmArea[1], manualOperationCms := #manualOperationCms[22], twoWayAcutor := #twoWayAcutor[2], Status => #Status[22], errorID => #errorID[22])
   END_RUNG
   RUNG wire#powerrail
      { S7_Templates := "SrcType := Int" } LE_Contact(in1 := #tempUpperBoundTwoWayAct, in2 := 2)
      JumpCoil( end )
   END_RUNG
   // the same network as SCL:
   "ManOperationCm_typeTwoWayActuatorInterface"(disableUnit := #disableUnit,
                           manualOperationEm := #manualOperationEm,
                           manualOperationEmArea := #manualOperationEmArea[1],
                           manualOperationCms := #manualOperationCms[22],
                           twoWayAcutor := #twoWayAcutor[2],
                           Status => #Status[22],
                           errorID => #errorID[22]);
   IF #tempUpperBoundTwoWayAct <= 2 THEN GOTO end; END_IF;
END_REGION

